							(* predefine rear side *)
							MachineCtrl.ProcessTemp.ActualJobData.SpecialTooth.VarioTooth.Distances.RearPos[0,0]	:=	1;
							MachineCtrl.ProcessTemp.ActualJobData.SpecialTooth.VarioTooth.Distances.RearPos[0,1]	:=	2;
							MachineCtrl.ProcessTemp.ActualJobData.SpecialTooth.VarioTooth.Distances.RearPos[1,0]	:=	3;
							MachineCtrl.ProcessTemp.ActualJobData.SpecialTooth.VarioTooth.Distances.RearPos[1,1]	:=	4;
							MachineCtrl.ProcessTemp.ActualJobData.SpecialTooth.VarioTooth.Distances.RearPos[2,0]	:=	5;
							MachineCtrl.ProcessTemp.ActualJobData.SpecialTooth.VarioTooth.Distances.RearPos[2,1]	:=	6;
							MachineCtrl.ProcessTemp.ActualJobData.SpecialTooth.VarioTooth.Distances.RearPos[3,0]	:=	7;
							MachineCtrl.ProcessTemp.ActualJobData.SpecialTooth.VarioTooth.Distances.RearPos[3,1]	:=	8;
							MachineCtrl.ProcessTemp.ActualJobData.SpecialTooth.VarioTooth.Distances.RearPos[4,0]	:=	9;
							MachineCtrl.ProcessTemp.ActualJobData.SpecialTooth.VarioTooth.Distances.RearPos[4,1]	:=	10;
							MachineCtrl.ProcessTemp.ActualJobData.SpecialTooth.VarioTooth.Distances.RearPos[5,0]	:=	11;
							MachineCtrl.ProcessTemp.ActualJobData.SpecialTooth.VarioTooth.Distances.RearPos[5,1]	:=	0;

							IF	( VarioCtrEnd < 5 )
								THEN
									MachineCtrl.ProcessTemp.ActualJobData.SpecialTooth.VarioTooth.Distances.RearPos[VarioCtrEnd,1]	:=	0;
							END_IF;

							FOR 	VarioCtr := 0 TO VarioCtrEnd
									DO
										VarioCtrFront1	:=	MachineCtrl.ProcessTemp.ActualJobData.SpecialTooth.VarioTooth.Distances.FrontPos[VarioCtr,0];
										VarioCtrFront2	:=	MachineCtrl.ProcessTemp.ActualJobData.SpecialTooth.VarioTooth.Distances.FrontPos[VarioCtr,1];
										VarioCtrRear1	:=	MachineCtrl.ProcessTemp.ActualJobData.SpecialTooth.VarioTooth.Distances.RearPos[VarioCtr,0];
										VarioCtrRear2	:=	MachineCtrl.ProcessTemp.ActualJobData.SpecialTooth.VarioTooth.Distances.RearPos[VarioCtr,1];

										MachineCtrl.ProcessTemp.ActualJobData.SpecialTooth.VarioTooth.Distances.Front[VarioCtr]	:=
																															VarioToothPitch[VarioCtrFront1] +
																															VarioToothPitch[VarioCtrFront2];

										MachineCtrl.ProcessTemp.ActualJobData.SpecialTooth.VarioTooth.Distances.Rear[VarioCtr]	:=
																															VarioToothPitch[VarioCtrRear1] +
																															VarioToothPitch[VarioCtrRear2];
							END_FOR;
						END_IF;
				END_IF;

				(*Transition*)
				IF	StepAction AND
					( RTrigNextStep.Q OR
					ContinousMode )
					THEN
						StepNew			:= 	1295;
						NextStepPulse	:=	FALSE;

						(* zero is the first element *)
						VarioCtr			:=	-1;
				END_IF;

	(*----------------------------------------------Calc Velocity For Automatic Process--------------------------------------------------*)

	1295:		(* action:   *)
					IF	StepActionImPulse
						THEN
							(* calc sawblade circumference *)
								SBCircumference				:=	ActualSawBlade.Diameter*PI;
								(* max feedrate chip breaker  *)
								ChipBreakerAutoXAxisMaxVelo	:=	45.0;
							(* calc velo x-axis degree/s *)
								ChipBreakerAutoVeloTemp		:=	( 360.0 * ChipBreakerAutoXAxisMaxVelo ) / SBCircumference;
								ChipBreakerXAxisVelo			:=	ChipBreakerAutoVeloTemp	;
					END_IF;

					(*Transition*)
					IF	StepAction  AND
						(NOT StepActionImPulse)
						THEN
							StepNew		:=	1297;	(*Switch On Cooling *)
					END_IF;
	(*--------------------------------------------------------Switch On Cooling ---------------------------------------------------------------*)
	1297:			(*Action*)
					IF	StepActionImPulse
						THEN
							MachineCtrl.Peripheral.ChipBreaker.Auto.Cooling.CmdOn	:=	TRUE;
							MachineCtrl.Peripheral.ChipBreaker.Auto.Cooling.CmdOff	:=	FALSE;
					END_IF;
					(*Transition*)
					IF	StepAction AND
						(NOT StepActionImPulse) AND
						MachineCtrl.State.ChipBreaker.Auto.Cooling.IsActive AND
						(NOT MachineCtrl.Peripheral.ChipBreaker.Auto.Cooling.CmdOn )
						THEN
							StepNew		:=	1300;	(*Start Process*)
					END_IF;


	(*--------------------------------------------------------------------Z-Axis Upfeed-------------------------------------------------------------*)
	1300:			(*Action*)
					IF	StepActionImPulse
						THEN
							MachineCtrl.Peripheral.ChipBreaker.Auto.DustFan.CmdOn			:=	TRUE;
							PauseAvailable												:=	TRUE;
							(*Is Demo Mode Active?*)
						(*	IF	UI.MachineSpecification.Base.DemoMode
								THEN
									ZAxisUpfeedMM	:=	-  ZAxisUpfeedMM - 1;
							END_IF;	*)
						(* set axis state for check *)
							AxisState													:=	STATE_WAIT_NEWOPERATION;
						(*	ZAxisUpfeedMM												:=	ActualJob.Infeed.TotalInfeed; *)
							ZAxisUpfeedPosition											:=	ZAxisStartPosition - (2* ZAxisUpfeedMM) ;
							ActualInfeed													:=	ActualRevolutions * MachineCtrl.ProcessTemp.ActualJobData.Job.Infeed.PartialInfeed;

							IF	( ActualJob.FeedRate.Override <= 0 )
								THEN
									ActualJob.FeedRate.Override	:=	1;
							END_IF;

							AxisCtrl[AxisNo.ZAxis].Command.OperationMode.CmdMoveAbsolut	:=	TRUE;
							AxisCtrl[AxisNo.ZAxis].Command.NominalValue.PositionMoveAbsolut	:=	ZAxisStartPosition - ZAxisUpfeedMM - 0.7;			(*= ZAxisUpfeedPosition*)
							AxisCtrl[AxisNo.ZAxis].Command.NominalValue.VeloMoveAbsolut	:=	ActualJob.FeedRate.Nominal *
																							ActualJob.FeedRate.Override;					(* velocity downfeed y-axis *)
							AxisCtrl[AxisNo.ZAxis].Command.ExternalControl.override			:=	100;
					END_IF;

					(* transition:  *)
					IF	StepAction AND
						(NOT StepActionImPulse) AND
						(* status y-axis *)
							Axis[AxisNo.ZAxis].Status.StandStill AND
							Axis[AxisNo.ZAxis].Status.InTargetPosition AND
							( AxisCtrl[AxisNo.ZAxis].feedback.state.ActualFbState = AxisState )
						THEN
							 StepNew			:= 	1305; 								(* Z-Axis Moves Down   *)
					END_IF;

	(*---------------------------------------------------------Wait For User Interaction--------------------------------------------------------------*)
		1305:		IF	StepActionImpulse
						THEN
							NextStepPulse	:=	TRUE;
					END_IF;
	
					IF	StepAction AND
						( RTrigNextStep.Q OR
						ContinousMode )
						THEN
							StepNew			:= 	1310;
							NextStepPulse	:=	FALSE;
					END_IF;

	(*--------------------------------------------------------------- Z-Axis Moves Down ---------------------------------------------------------------- *)
	1310:			(*Action*)
					IF	StepActionImPulse
						THEN
							AxisCtrl[AxisNo.ZAxis].Command.OperationMode.CmdMoveAbsolut		:=	TRUE;
							AxisCtrl[AxisNo.ZAxis].Command.NominalValue.PositionMoveAbsolut		:= 	ZAxisStartPosition ;
							AxisCtrl[AxisNo.ZAxis].Command.NominalValue.VeloMoveAbsolut		:=	3.5;
					END_IF;

					(* transition:  *)

					IF	StepAction AND
						(NOT StepActionImPulse) AND
						(* Complete movement *)
						(NOT AxisCtrl[AxisNo.ZAxis].Command.OperationMode.CmdMoveAbsolut)
						THEN
							IF	ChipBreakerfr				(*ChipBreaekerIsInFrontPosition*)
								THEN
									NominalTeeth	:=	MachineCtrl.ProcessTemp.ActualOrderStackBuffer.ActualOrder.SawBlade.NumberOfTeeth / 2;
									ActualRevolutions	:=	0;

								ELSIF	 ChipBreakerRe	(*ChipBreaekerIsInRearPosition*)
									THEN
											NominalTeeth	:=	MachineCtrl.ProcessTemp.ActualOrderStackBuffer.ActualOrder.SawBlade.NumberOfTeeth;

											ActualRevolutions	:=	1;
								END_IF;

							ActualTeeth		:=	ActualTeeth + 1;

							IF	( ActualTeeth >= NominalTeeth )
								THEN
										StepNew				:= 	10000;			(*Finish The Process*)
									ELSE
										StepNew				:= 	1350;	(*Actual Teeth <> Nominal Teeth*)
							END_IF;
								ActualInfeed			:=	ActualRevolutions * MachineCtrl.ProcessTemp.ActualJobData.Job.Infeed.PartialInfeed;
								PartialInfeed			:=	MachineCtrl.ProcessTemp.ActualJobData.Job.Infeed.PartialInfeed;
					END_IF;

	(* ---------------------------------------------------------- move x-axis ccw 2 teeth --------------------------------------------------------- *)
	1350:			(* action: *)
					IF	StepActionImPulse
						THEN
							AxisCtrl[AxisNo.XAxis].Command.OperationMode.CmdMoveAbsolut		:=	TRUE;

							IF	MachineCtrl.ProcessTemp.ActualJobData.SpecialTooth.VarioTooth.IsActive
								THEN
									VarioCtr	:=	VarioCtr + 1;

									IF	ChipBreakerRe	(*Input Variable To set The Side *)
										THEN
											AxisCtrl[AxisNo.XAxis].Command.NominalValue.PositionMoveAbsolut			:= 	Axis[AxisNo.XAxis].NcToPlc.ActPos +
																													MachineCtrl.ProcessTemp.ActualJobData.SpecialTooth.VarioTooth.Distances.Rear[VarioCtr];

										ELSIF	ChipBreakerFr
											THEN
												AxisCtrl[AxisNo.XAxis].Command.NominalValue.PositionMoveAbsolut		:= 	Axis[AxisNo.XAxis].NcToPlc.ActPos +
																													MachineCtrl.ProcessTemp.ActualJobData.SpecialTooth.VarioTooth.Distances.Front[VarioCtr];
									END_IF;

									IF	VarioCtr = VarioCtrEnd
										THEN
											VarioCtr	:=	-1;
									END_IF;

								ELSE
								(*Varion Is Inactive*)
								IF	MachineCtrl.ProcessTemp.ActualJobData.SpecialTooth.TKCompensationActive
									THEN
										IF	NoOfActTeethCompensation <> 1
											THEN
											XAxisNextPosition	:=		 Axis[AxisNo.XAxis].NcToPlc.ActPos
															         + ( 2*DegPerTeeth -
																 AxisPhasingCAM.CbaTeethDiff[NoOfActTeethCompensation] -
																 AxisPhasingCAM.CbaTeethDiff[NoOfActTeethCompensation -1] );
											ELSE
											XAxisNextPosition	:=		 Axis[AxisNo.XAxis].NcToPlc.ActPos
															         + ( 2*DegPerTeeth -
																 AxisPhasingCAM.CbaTeethDiff[1] -
																 AxisPhasingCAM.CbaTeethDiff[UI.Order.SawBlade.NumberOfTeeth] );
										END_IF;

										AxisCtrl[AxisNo.XAxis].Command.NominalValue.PositionMoveAbsolut		:= 	XAxisNextPosition;
									ELSE
										AxisCtrl[AxisNo.XAxis].Command.NominalValue.PositionMoveAbsolut		:= 	Axis[AxisNo.XAxis].NcToPlc.ActPos + ( 2 *	DegPerTeeth );
								END_IF;
							END_IF;

							AxisCtrl[AxisNo.XAxis].Command.NominalValue.VeloMoveAbsolut					:=	ChipBreakerXAxisVelo;
							AxisCtrl[AxisNo.XAxis].Command.ExternalControl.override							:=	100;
					END_IF;

					(* transition:  *)

					IF	StepAction AND
						(NOT StepActionImPulse) AND
						(* Complete movement *)
						NOT AxisCtrl[AxisNo.XAxis].Command.OperationMode.CmdMoveAbsolut
						THEN

						IF	ActualTeeth < NominalTeeth
							THEN
								NoOfActTeethCompensation		:=		NoOfActTeethCompensation   -   2 ;
								ELSIF
									(ActualTeeth = NominalTeeth)
								THEN
								;
						END_IF;

						IF	NoOfActTeethCompensation <0
							THEN
								NoOfActTeethCompensation	:=	TO_INT(UI.Order.SawBlade.NumberOfTeeth) + NoOfActTeethCompensation ;
						END_IF;

						IF	NoOfActTeethCompensation =0
							THEN
								NoOfActTeethCompensation	:=	TO_INT(UI.Order.SawBlade.NumberOfTeeth)  ;
						END_IF;

							IF 	(XAxisEndPos =AxisCtrl[AxisNo.XAxis].Command.NominalValue.PositionMoveAbsolut)		(*Check If X Reached The End Position*)
								THEN
									ContinousMode	:=	FALSE;
									StepNew		:= 	9000;														(*Check  side  finished*)
									ELSE
										IF	PauseRequested
											THEN
												ContinousMode	:=	FALSE;
												PauseAvailable	:=	FALSE;
												StepNew			:= 	30050;										(* -> pause Routine *)
											ELSE
												StepNew			:=	1300;										(*Z-Axis Upfeed*)
										END_IF;
							END_IF;
					END_IF;

	(*---------------------------------------------------------Wait For User Interaction----------------------------------------------------------*)
	9000:		IF	StepActionImpulse
					THEN
						NextStepPulse	:=	TRUE;
				END_IF;

				IF	StepAction AND
					( RTrigNextStep.Q OR
					ContinousMode )
					THEN
						StepNew			:= 	10000;
						NextStepPulse	:=	FALSE;
				END_IF;
	(*---------------------------------------------------------------End Front Side -----------------------------------------------------------------*)
	10000:		(*Transition*)
				IF	ChipBreakerFr AND
					(NOT ChipBreakerRe)
					THEN
					StepNew		:=	15000;				(*END_Front Side  *)
					XaxisEndPOsFront	:=	Axis[AxisNo.XAxis].NcToPlc.ActPos;
						ELSIF	ChipBreakerRe
					THEN
						StepNew		:=	10050;	(*Proceed to the End of Process*)
						MachineCtrl.Peripheral.ChipBreaker.Auto.DustFan.CmdOn	:=	FALSE;
				END_IF;
	(*-------------------------------------------------------Wait For User Interaction----------------------------------------------------------*)
	10050:
				IF	StepActionImpulse
					THEN
						NextStepPulse	:=	TRUE;
				END_IF;

				IF	StepAction AND
					( RTrigNextStep.Q OR
					ContinousMode )
					THEN
						StepNew			:= 	10100;
						NextStepPulse	:=	FALSE;
				END_IF;

	(* ----------------------------------------------------------- disable  Turbine  -------------------------------------------------------------- *)
	10100:		(* action *)
					IF	StepActionImPulse
						THEN
							MachineCtrl.Peripheral.ChipBreaker.Auto.Turbine.CmdOn	:=	FALSE;
							MachineCtrl.Peripheral.ChipBreaker.Auto.Turbine.CmdOff	:=	TRUE;
					END_IF;

					(* transition *)
					IF	StepAction AND
						( NOT StepActionImPulse ) AND
						( NOT MachineCtrl.Peripheral.ChipBreaker.Auto.Turbine.CmdOn )
						THEN
							StepNew		:=	10120;		(*Switch Off Fan*)
					END_IF;
	(*----------------------------------------------------------Switch Off Cooling -------------------------------------------------------*)
	10120:
					(*Action*)
					IF	StepActionImPulse
						THEN
							MachineCtrl.Peripheral.ChipBreaker.Auto.Cooling.CmdOn	:=	FALSE;
							MachineCtrl.Peripheral.ChipBreaker.Auto.Cooling.CmdOff	:=	TRUE;
					END_IF;
					(*Transition*)
					IF	StepAction AND
						(NOT StepActionImPulse) AND
						MachineCtrl.State.ChipBreaker.Auto.Cooling.IsInactive  AND
						(NOT MachineCtrl.Peripheral.ChipBreaker.Auto.Cooling.CmdOff )
						THEN
							StepNew		:=	10150;	(* ->Release Clamping *)
					END_IF;
	(*--------------------------------------------------Wait For User Interaction------------------------------------------------------------*)
	10150:		IF	StepActionImpulse
					THEN
						NextStepPulse	:=	TRUE;
				END_IF;

				IF	StepAction AND
					( RTrigNextStep.Q OR
					ContinousMode )
					THEN
						StepNew			:= 	10200;			(*Release Clamping*)
						NextStepPulse	:=	FALSE;
				END_IF;

	(*--------------------------------------------------------- Release clamping ------------------------------------------------------------- *)
	10200:		(* action *)
					IF	StepActionImPulse
						THEN
							MachineCtrl.Peripheral.ChipBreaker.Auto.Clamping.CmdClose	:=	FALSE;
							MachineCtrl.Peripheral.ChipBreaker.Auto.Clamping.CmdOpen	:=	TRUE;
					END_IF;

					(* transition:  *)
					IF	StepAction AND
						(NOT StepActionImPulse) AND
						(* clamping is opene *)
						MachineCtrl.State.ChipBreaker.Auto.Clamping.IsReleased
						THEN
							StepNew	:= 	10450;										(*Z-Axis-->Ref Pos & Saw Blade Bracket To Home Pos*)
					END_IF;
	(*--------------------------------------------Wait For User Interaction-------------------------------------------------------*)
	10450:		IF	StepActionImpulse
					THEN
						NextStepPulse	:=	TRUE;
				END_IF;

				IF	StepAction AND
					( RTrigNextStep.Q OR
					ContinousMode )
					THEN
						StepNew			:= 	10500;
						NextStepPulse	:=	FALSE;
				END_IF;
	(* ------------------------------------------------------------ sfc finished ---------------------------------------------------------- *)
	10500:		(*Action*)
					IF	 StepActionImPulse AND
						(NOT  AxisCtrl[AxisNo.ZAxis].feedback.state.DriveManagment.InHandoverPositionWindow)
						THEN
							(* Z-axis - move absolute *)
							AxisCtrl[AxisNo.ZAxis].Command.OperationMode.CmdPowerOn			:=	TRUE;
							AxisCtrl[AxisNo.ZAxis].Command.OperationMode.CmdJogHandwheel 		:=	FALSE;
							AxisCtrl[AxisNo.ZAxis].Command.OperationMode.CmdMoveAbsolut		:=	TRUE;
							AxisCtrl[AxisNo.ZAxis].Command.OperationMode.CmdCamming			:=	FALSE;
							AxisCtrl[AxisNo.ZAxis].Command.NominalValue.VeloMoveAbsolut		:=	100;
							AxisCtrl[AxisNo.ZAxis].Command.NominalValue.PositionMoveAbsolut		:=	UI.MachineSpecification.PeripheralBasic.Axis.Positions.HandOver;
							MachineCtrl.Peripheral.ChipBreaker.Auto.DustFan.CmdOn				:=	FALSE;
					END_IF;

					(*Transition : Is Z- Axis In Handover Pos?*)

					IF     	StepAction AND
					   	 (NOT StepActionImPulse) AND
						 AxisCtrl[AxisNo.ZAxis].feedback.state.DriveManagment.InHandoverPositionWindow
						THEN
							StepNew			:=	10700;							(*SB Support Bracket To Home Pos*)
							ContinousMode	:=	FALSE;
					END_IF;
	(*----------------------------------------------Wait For User Interaction------------------------------------------------*)
	10700:
					IF	StepAction AND
						NOT StepActionImPulse
						THEN
							IF	Stepper  AND
								(NOT CbaPneumatic)
								THEN
									IF	(NOT UI.MachineSpecification.Base.DemoMode)
										THEN
											StepNew		:=	10750;
										ELSE
											StepNew		:=	11000;
									END_IF;

								ELSIF	(NOT Stepper)  AND
										 CbaPneumatic
								THEN
									IF	(NOT UI.MachineSpecification.Base.DemoMode)
										THEN
											StepNew		:=	10800;
										ELSE
											StepNew		:=	11000;
									END_IF;
							END_IF;
					END_IF;

	(*----------------------------------------------------Move A-Stepper To Ref position------------------------------- *)
	10750:
				IF 	StepActionImpulse
					THEN
						AxisCtrl[AxisNo.AAxis].Command.OperationMode.CmdJog				:=	TRUE;
						AxisCtrl[AxisNo.AAxis].Command.ExternalControl.Override				:=	100;
						AxisCtrl[AxisNo.AAxis].Command.NominalValue.VeloJog				:=	0.5;
						IF	(MachineCtrl.State.ChipBreaker.Auto.AaxisActualPos <=   UI.MachineSpecification.PeripheralOptional.ChipBreaker.Notch.SBEdgeOffset)
							THEN
								AxisCtrl[AxisNo.AAxis].Command.ExternalControl.StartMinus				:=	TRUE;
								AxisCtrl[AxisNo.AAxis].Command.ExternalControl.StartPlus				:=	FALSE;;
							ELSE
								AxisCtrl[AxisNo.AAxis].Command.ExternalControl.StartMinus				:=	FALSE;
								AxisCtrl[AxisNo.AAxis].Command.ExternalControl.StartPlus				:=	TRUE;;
						END_IF;
						StartMonitoringAaxis												:=	TRUE;
				END_IF;
				(*Transition*)
				IF 	StepAction AND
					(NOT  StepActionImpulse) AND
					(MachineCtrl.State.ChipBreaker.Auto.AaxisActualPos >=  ( UI.MachineSpecification.PeripheralOptional.ChipBreaker.Notch.SBEdgeOffset  - AaxisTolerenceSlow)) AND
					(MachineCtrl.State.ChipBreaker.Auto.AaxisActualPos <=  (  UI.MachineSpecification.PeripheralOptional.ChipBreaker.Notch.SBEdgeOffset + AaxisTolerenceSlow))
					THEN
						AxisCtrl[AxisNo.AAxis].Command.ExternalControl.StartMinus				:=	FALSE;
						AxisCtrl[AxisNo.AAxis].Command.ExternalControl.StartPlus				:=	FALSE;;
						StepNew			:=	11000;
				END_IF;

	(*----------------------------------------------------Move  Cylindre To Front Position------------------------------- *)

	10800:		(*Action*)
				IF 	StepActionImpulse AND
					(NOT MachineCtrl.State.ChipBreaker.Auto.TurbinePosition.InFrontPosition)
					THEN
						MachineCtrl.Peripheral.ChipBreaker.Auto.TurbinePosition.CmdBackward	:=	FALSE;
						MachineCtrl.Peripheral.ChipBreaker.Auto.TurbinePosition.CmdForward	:=	TRUE;
				END_IF;
				(*Transition*)
				IF 	StepAction AND
					(NOT StepActionImpulse) AND
					(NOT MachineCtrl.Peripheral.ChipBreaker.Auto.TurbinePosition.CmdForward) AND
					 MachineCtrl.State.ChipBreaker.Auto.TurbinePosition.InFrontPosition
					THEN
							StepNew		:=	11000;
				END_IF;
	(*--------------------------------------CBA Swivel UnitTo Home Position----------------------------------------*)
	11000:		(*Action*)
					IF	StepActionImPulse
						THEN
							MachineCtrl.Peripheral.ChipBreaker.Auto.SwivelUnit.CmdHomePos	:=	TRUE;
							MachineCtrl.Peripheral.ChipBreaker.Auto.SwivelUnit.CmdWorkPos	:=	FALSE;
							StartMonitoringAaxis											:=	FALSE;
					END_IF;
					(*Transition*)
					IF 	StepAction AND
						(NOT StepActionImPulse) AND
						MachineCtrl.State.ChipBreaker.Auto.SwivelUnit.InHomePosition
						THEN
							StepNew		:=	11010;	(*Wait for New Operation*)
					END_IF;

	(*----------------------------------------------------Wait For User Interaction-----------------------------------------------*)
	11010:
					IF	StepActionImpulse
						THEN
							NextStepPulse	:=	TRUE;
					END_IF;
	
					IF	StepAction AND
						( RTrigNextStep.Q OR
						ContinousMode )
						THEN
							StepNew			:= 	15000;
							NextStepPulse	:=	FALSE;
					END_IF;
	(*---------------------------------------Step 10 : Wait for New Operation-------------------------------------------*)

	15000:		(* transition *)
					IF	StepAction AND
						(NOT StepActionImPulse)
							THEN
								IF 	ChipBreakerRe
									THEN
										StepNew				:= 	16000;			(*Wait For New Operation*)
										MachineCtrl.Peripheral.ChipBreaker.Auto.LowSpeedMonitoring.IsDeactivated	:=	FALSE;
										Done				:=	TRUE;
										Start					:=	FALSE;
										ChipBreakerFr		:=	TRUE;
										ChipBreakerRe		:=	FALSE;
									ELSIF 	ChipBreakerFr
										THEN
										ChipBreakerFr	:=	FALSE;
										ChipBreakerRe	:=	TRUE;
										IF	Stepper AND
											(NOT CbaPneumatic)
											THEN
												StepNew			:= 	950;		(*Start With The Rear Side*)
											ELSIF	CbaPneumatic AND
													(NOT Stepper)
											THEN
												StepNew			:= 	990;
										END_IF;
										Done	:=	FALSE;
								END_IF;
					END_IF;

	(*---------------------------------------Wait For User Interaction---------------------------------------------------------*)
	16000:		IF	StepActionImpulse
					THEN
						NextStepPulse	:=	TRUE;
				END_IF;

				IF	StepAction AND
					( RTrigNextStep.Q OR
					ContinousMode )
					THEN
						StepNew			:= 	10;
						NextStepPulse	:=	FALSE;
				END_IF;

	(*--##################################---ERROR-###################################- *)

	25000:		(*Action*)
				IF	 StepActionImPulse
					THEN
						MachineCtrl.Peripheral.ChipBreaker.Auto.DustFan.CmdOn			:=	FALSE;
						AxisCtrl[AxisNo.AAxis].Command.ExternalControl.StartPlus			:=	FALSE;
						AxisCtrl[AxisNo.AAxis].Command.ExternalControl.StartMinus			:=	FALSE;		(*Stop Moving   A-Axis*)
						ErrorOut			:=	TRUE;
				END_IF;
				(*Transition*)

				IF 	StepAction AND
					(NOT StepActionImPulse)
					THEN
						StepNew		:=	0;
						ErrorOut		:=	FALSE;
				END_IF;
	(* ####################################### pause sfc ################################ *)

	(*-----------------------------------------------------------Wait For User Interaction------------------------------------------------*)
	30050:
				 IF	StepActionImpulse
					THEN
						NextStepPulse	:=	TRUE;
				END_IF;

				IF	StepAction AND
					( RTrigNextStep.Q OR
					ContinousMode )
					THEN
						StepNew			:= 	30100;		(*Release Clamping*)
						NextStepPulse	:=	FALSE;
				END_IF;

	(*--------------------------------------------------------------Release Clamping-----------------------------------------------------*)
	30100:
					(*Action*)
				IF	StepActionImPulse
					THEN
						MachineCtrl.Peripheral.ChipBreaker.Auto.Clamping.CmdClose	:=	FALSE;
						MachineCtrl.Peripheral.ChipBreaker.Auto.Clamping.CmdOpen	:=	TRUE;
				END_IF;

				(* transition:  *)

				IF	StepAction AND
					(NOT StepActionImPulse) AND
					MachineCtrl.State.ChipBreaker.Auto.Clamping.IsReleased
					THEN
						StepNew	:= 	30200;					(*Z Axis Move   down 100 MM*)
				END_IF;
	(* ----------------------------------------------------- wait for user interaction  ---------------------------------------------------- *)
	30200:
				IF	StepActionImpulse
					THEN
						NextStepPulse	:=	TRUE;
				END_IF;

				IF	StepAction AND
					( RTrigNextStep.Q OR
					ContinousMode )
					THEN
						StepNew			:= 	30250;
						NextStepPulse	:=	FALSE;
				END_IF;
	(* ------------------------------------------------- sfc Paused: move Z-axisDown ------------------------------------------------- *)

	30250	:	(* action: move z-axis down  *)
				IF	StepActionImPulse
					THEN
					(* set axis state for check *)
						AxisState	:=	STATE_WAIT_NEWOPERATION;
					(* move y-axis to reference point *)
						AxisCtrl[AxisNo.ZAxis].Command.OperationMode.CmdPowerOn					:=	TRUE;
						AxisCtrl[AxisNo.ZAxis].Command.OperationMode.CmdMoveAbsolut				:=	TRUE;
						AxisCtrl[AxisNo.ZAxis].Command.NominalValue.PositionMoveAbsolut				:=	Axis[AxisNo.ZAxis].NcToPlc.ActPos	+100;
						AxisCtrl[AxisNo.ZAxis].Command.NominalValue.VeloMoveAbsolut				:=	30;
						MachineCtrl.Peripheral.ChipBreaker.Auto.DustFan.CmdOn						:=	FALSE;
				END_IF;

				(* transition *)
				IF	StepAction AND
					(NOT StepActionImPulse) AND
					(* status Z-axis *)
					Axis[AxisNo.ZAxis].Status.StandStill AND
					Axis[AxisNo.ZAxis].Status.InTargetPosition AND
					( NOT AxisCtrl[AxisNo.ZAxis].Command.OperationMode.CmdMoveAbsolut ) AND
					( AxisCtrl[AxisNo.ZAxis].feedback.state.ActualFbState = AxisState )
					THEN
						StepNew		:= 30300;															(*Turbine Off*)
				END_IF;

	(* ---------------------------------------------------- wait for user interaction  ------------------------------------------------------------ *)
	30300:		IF	StepActionImpulse
					THEN
						NextStepPulse	:=	TRUE;
				END_IF;

				IF	StepAction AND
					( RTrigNextStep.Q OR
					ContinousMode )
					THEN
						StepNew			:= 	30350;	(*Turbine Off*)
						NextStepPulse	:=	FALSE;
				END_IF;

	(* --------------------------------------------------------------- Turbine Off --------------------------------------------------------------------- *)
	30350	:	(* action:   *)
				IF	StepActionImPulse
					THEN
						MachineCtrl.Peripheral.ChipBreaker.Auto.Turbine.CmdOn	:=	FALSE;
						MachineCtrl.Peripheral.ChipBreaker.Auto.Turbine.CmdOff	:=	TRUE;
				END_IF;
				(* transition: *)
				IF	StepAction AND
					( NOT StepActionImPulse ) AND
					( NOT MachineCtrl.Peripheral.ChipBreaker.Auto.Turbine.CmdOn )AND
					(NOT MachineCtrl.State.ChipBreaker.Auto.Turbine.IsActive)			(*Turbine Is Inactive*)
					THEN
							StepNew		:=	30370	;
				END_IF;

	(*-------------------------------------------------------Switch Off Cooling --------------------------------------------------------------------*)
	30370:
				(*Action*)
				IF	StepActionImPulse
					THEN
						MachineCtrl.Peripheral.ChipBreaker.Auto.Cooling.CmdOn	:=	FALSE;
						MachineCtrl.Peripheral.ChipBreaker.Auto.Cooling.CmdOff	:=	TRUE;
				END_IF;
				(*Transition*)
				IF	StepAction AND
					(NOT StepActionImPulse) AND
					MachineCtrl.State.ChipBreaker.Auto.Cooling.IsInactive  AND
					(NOT MachineCtrl.Peripheral.ChipBreaker.Auto.Cooling.CmdOff )
					THEN
						StepNew		:=	30400;	(* ->deactivate axis x/z *)
				END_IF;
	(* ------------------------------------------------------ wait for user interaction  -------------------------------------------------------------- *)
	30400:
				IF	StepActionImpulse
					THEN
						NextStepPulse	:=	TRUE;
				END_IF;

				IF	StepAction AND
					( RTrigNextStep.Q OR
					ContinousMode )
					THEN
						StepNew			:= 	30450;
						NextStepPulse	:=	FALSE;
				END_IF;
	(*---------------------------------------------------------------Desable X/Z Axis-----------------------------------------------------------------*)
	30450:
				(* action:   *)
				IF	StepActionImPulse
					THEN
						(* set axis state for check *)
							AxisState	:=	STATE_INIT;
						(* x-axis - disable *)
							AxisCtrl[AxisNo.XAxis].Command.OperationMode.CmdPowerOn			:=	FALSE;
							AxisCtrl[AxisNo.XAxis].Command.OperationMode.CmdMoveAbsolut		:=	FALSE;
							AxisCtrl[AxisNo.XAxis].Command.OperationMode.CmdCamming			:=	FALSE;
						(* z-axis - disable *)
							AxisCtrl[AxisNo.ZAxis].Command.OperationMode.CmdPowerOn			:=	FALSE;
							AxisCtrl[AxisNo.ZAxis].Command.OperationMode.CmdMoveAbsolut		:=	FALSE;
							AxisCtrl[AxisNo.ZAxis].Command.OperationMode.CmdCamming			:=	FALSE;
				END_IF;
				(* transition:  *)
				IF	StepAction AND
					(NOT StepActionImPulse) AND
					(* status x-axis *)
						Axis[AxisNo.XAxis].Status.Disabled AND
						( AxisCtrl[AxisNo.XAxis].feedback.state.ActualFbState = AxisState ) AND
					(* status z-axis *)
						Axis[AxisNo.ZAxis].Status.Disabled AND
						( AxisCtrl[AxisNo.ZAxis].feedback.state.ActualFbState = AxisState )
						THEN
							StepNew		:= 	30460;			(*User Interaction*)
				END_IF;
	(* ------------------------------------------------------------- wait for user interaction  -------------------------------------------------------- *)
	30460:
				IF	StepActionImpulse
					THEN
						NextStepPulse	:=	TRUE;
				END_IF;

				IF	StepAction AND
					( RTrigNextStep.Q OR
					ContinousMode )
					THEN
						StepNew			:= 	30470;		(* -> Activate Safety State*)
						NextStepPulse	:=	FALSE;
				END_IF;
	(* -------------------------------------------------------- Activate Safety State -------------------------------------------------------------- *)
	30470:				(*Action*)
				IF	StepActionImPulse
					THEN
					(* Enable safe state  *)
						MachineCtrl.Peripheral.SafetyState.CmdActivate	:=	TRUE;
						MachineCtrl.State.GrindingWheel.PauseIsActive	:=	TRUE;
				END_IF;
				(* transition:  *)
				IF	StepAction AND
					(NOT StepActionImPulse) AND
					(* state safety state *)
					( NOT MachineCtrl.Peripheral.SafetyState.CmdActivate ) AND
					MachineCtrl.state.SafetyState.unit.IsActive
					THEN
						StepNew		:=	30500;
				END_IF;

	(*--------------------------------------------------------------------Set Event----------------------------------------------------------------------*)
				(*Action*)
	30500:
				IF	StepActionImPulse
					THEN
				(* set Event *)
						MachineCtrl.ProcessControl.Event.No		:=	EvNoStartStop;
						MachineCtrl.ProcessControl.Event.En		:=	TRUE;
						MachineCtrl.ProcessControl.Event.SId	:=	EvEventSourceId;
						MachineCtrl.ProcessControl.Event.Class	:=	TcEventClassMessage;
						MachineCtrl.Peripheral.Buzzer.Unit.CmdOn:=	TRUE;
				END_IF;
				(*Transition*)
				IF	StepAction AND
					(NOT StepActionImPulse)
					THEN
						StepNew		:=	30520;
				END_IF;

	(* --------------------------------------------------------- wait for user interaction  ---------------------------------------------------------- *)
	30520:		IF	StepActionImpulse
					THEN
						NextStepPulse	:=	TRUE;
				END_IF;

				IF	StepAction AND
					( RTrigNextStep.Q OR
					ContinousMode )
					THEN
						MachineCtrl.Peripheral.ChipBreaker.Auto.DustFan.CmdOn					:=	FALSE;
						MachineCtrl.Peripheral.ChipBreaker.Auto.LowSpeedMonitoring.IsDeactivated	:=	FALSE;
						StepNew			:= 	30550;	(*Deactivate Safety  State *)
						NextStepPulse	:=	FALSE;
						Paused			:=	TRUE;
				END_IF;
	(* -----------------------------------------------------Deactivate Safety State---------------------------------------------------------- *)
	30550:			(* action:   *)
				IF	MachineCtrl.state.SafetyState.unit.IsActive
					THEN
						MachineCtrl.Peripheral.ChipBreaker.Auto.LowSpeedMonitoring.IsDeactivated	:=	FALSE;
						IF	MachineStateSharpenerDoorIsClosed AND
							AutomaticMode
							THEN
								(* Disable safe state  *)
								MachineCtrl.Peripheral.SafetyState.CmdDeactivate	:=	TRUE;
								MachineCtrl.State.GrindingWheel.PauseIsActive	:=	FALSE;
							ELSE
								(* Disable safe state  *)
								MachineCtrl.Peripheral.SafetyState.CmdDeactivate	:=	FALSE;
								MachineCtrl.Peripheral.SafetyState.CmdActivate	:=	TRUE;
								MachineCtrl.State.GrindingWheel.PauseIsActive	:=	TRUE;
						END_IF;
				END_IF;

				TONWaitSafetyStatePause( IN  	:=  	StepAction AND
												( NOT MachineCtrl.Peripheral.SafetyState.CmdDeactivate ) AND
												( NOT MachineCtrl.state.SafetyState.unit.IsActive ),
										 PT 	:= 	TIME#50ms);

				(* transition:  *)
				IF	StepAction AND
					(NOT StepActionImPulse) AND
					(* state safety state *)
						( NOT MachineCtrl.Peripheral.SafetyState.CmdDeactivate ) AND
						( NOT MachineCtrl.state.SafetyState.unit.IsActive ) AND
						TONWaitSafetyStatePause.Q (* AND
					StartSwitch *)
					THEN
						MachineCtrl.ProcessControl.Event.No		:=	0;
						MachineCtrl.ProcessControl.Event.En		:=	FALSE;
						StepNew								:= 	30600;	(*Turbine On*)
				END_IF;

	(* ----------------------------------------------------------- wait for user interaction  ------------------------------------------------ *)
	30600:		IF	StepActionImpulse
					THEN
						MachineCtrl.Peripheral.ChipBreaker.Auto.LowSpeedMonitoring.IsDeactivated	:=		TRUE;
						NextStepPulse	:=	TRUE;
				END_IF;

				IF	StepAction AND
					( RTrigNextStep.Q OR
					ContinousMode )
					THEN
						StepNew			:= 	30650;			(*Activate Turbine *)
						NextStepPulse	:=	FALSE;
				END_IF;

	(*------------------------------------------------------------------Turbine On--------------------------------------------------------------------*)
	30650:			(*Action*)
				IF	 StepActionImPulse
						THEN
							MachineCtrl.Peripheral.ChipBreaker.Auto.Turbine.CmdOn	:=	TRUE;
							MachineCtrl.Peripheral.ChipBreaker.Auto.Turbine.CmdOff	:=	FALSE;
				END_IF;
				(*Transition: Is the  Turbine On? *)
				IF	 StepAction 	AND
					 (NOT StepActionImPulse) AND
				    	  MachineCtrl.State.ChipBreaker.Auto.Turbine.IsActive
					THEN
						StepNew		:=	30660;		(*Switch On Cooling Fan*)
				END_IF;

	(*---------------------------------------------------- Switch On Cooling -------- --------------------------------------------------------------*)

	30660:
			(*Action*)
				IF	StepActionImPulse
					THEN
						MachineCtrl.Peripheral.ChipBreaker.Auto.Cooling.CmdOn	:=	TRUE;
						MachineCtrl.Peripheral.ChipBreaker.Auto.Cooling.CmdOff	:=	FALSE;
				END_IF;
				(*Transition*)
				IF	StepAction AND
					(NOT StepActionImPulse) AND
					MachineCtrl.State.ChipBreaker.Auto.Cooling.IsActive AND
					(NOT MachineCtrl.Peripheral.ChipBreaker.Auto.Cooling.CmdOn )
					THEN
						StepNew		:=	30670;	(*Start Process*)
				END_IF;

	(* ---------------------------------------------------- wait for user interaction  ------------------------------------------------------------ *)
	30670:
				IF	StepActionImpulse
					THEN
						NextStepPulse	:=	TRUE;
				END_IF;

				IF	StepAction AND
					( RTrigNextStep.Q OR
					ContinousMode )
					THEN
						StepNew			:= 	30680;			(*Open Clamping*)
						NextStepPulse	:=	FALSE;
				END_IF;
	(* ------------------------------------------------------- sfc Paused: Open Clamping ---------------------------------------------------- *)
	30680	:		(*Action*)
				IF	StepActionImPulse
					THEN
						MachineCtrl.Peripheral.ChipBreaker.Auto.Clamping.CmdClose	:=	FALSE;
						MachineCtrl.Peripheral.ChipBreaker.Auto.Clamping.CmdOpen	:=	TRUE;
				END_IF;
				(* transition:  *)
				IF	StepAction AND
					(NOT StepActionImPulse) AND
					MachineCtrl.State.ChipBreaker.Auto.Clamping.IsReleased
				THEN
						StepNew	:= 	30700;			(*Move Z To Start Pos*)
				END_IF;

	(* ----------------------------------------------------------- wait for user interaction  --------------------------------------------------------- *)
	30700:		IF	StepActionImpulse
					THEN
						NextStepPulse	:=	TRUE;
				END_IF;

				IF	StepAction AND
					( RTrigNextStep.Q OR
					ContinousMode )
					THEN
						StepNew			:= 	30710;
						NextStepPulse	:=	FALSE;
				END_IF;

	(*----------------------------------------------------------Move Z Axis To Start Pos-----------------------------------------------------------*)
	30710:
					(*Action*)
				IF	StepActionImPulse
				THEN
					AxisState	:=	STATE_WAIT_NEWOPERATION;
				(* Z-axis - move absolute *)
					AxisCtrl[AxisNo.ZAxis].Command.OperationMode.CmdPowerOn			:=	TRUE;
					AxisCtrl[AxisNo.ZAxis].Command.OperationMode.CmdJogHandwheel 		:=	FALSE;
					AxisCtrl[AxisNo.ZAxis].Command.OperationMode.CmdMoveAbsolut		:=	TRUE;
					AxisCtrl[AxisNo.ZAxis].Command.OperationMode.CmdCamming			:=	FALSE;
					AxisCtrl[AxisNo.ZAxis].Command.NominalValue.PositionMoveAbsolut		:=	ZAxisStartPosition;			(* Startposition y-axis *)
					AxisCtrl[AxisNo.ZAxis].Command.NominalValue.VeloMoveAbsolut		:=	15;						(* velocity Startpos z-axis *)
					AxisCtrl[AxisNo.ZAxis].Command.ExternalControl.override				:=	100;
				END_IF;

				(*Transition : Is /Z Axis in Start Position*)
				IF 	StepAction AND
					(NOT StepActionImPulse) AND
					(* status Z-axis *)
						Axis[AxisNo.ZAxis].Status.StandStill AND
						Axis[AxisNo.ZAxis].Status.InTargetPosition AND
						( NOT AxisCtrl[AxisNo.ZAxis].Command.OperationMode.CmdMoveAbsolut ) AND
						( AxisCtrl[AxisNo.ZAxis].feedback.state.ActualFbState = AxisState )
				THEN
					StepNew		:=	30800;		(*Clamping*)
				END_IF;

	(* ---------------------------------------------------- wait for user interaction  ------------------------------------------------------------- *)
	30800:
				IF	StepActionImpulse
					THEN
						NextStepPulse	:=	TRUE;
				END_IF;

				IF	StepAction AND
					( RTrigNextStep.Q OR
					ContinousMode )
					THEN
						StepNew			:= 	30860; (*Close Clamping*)
						NextStepPulse	:=	FALSE;
				END_IF;
	(*-----------------------------------------------------------------Close Klamping------------------------------------------------------------*)
	30860:
				(*Action*)
				IF	StepActionImPulse
					THEN
						MachineCtrl.Peripheral.ChipBreaker.Auto.Clamping.CmdClose	:=	TRUE;
						MachineCtrl.Peripheral.ChipBreaker.Auto.Clamping.CmdOpen	:=	FALSE;
				END_IF;

				WaitAfterPause(IN:=	StepAction AND
									(NOT StepActionImPulse) AND
									(* clamping is open *)
									MachineCtrl.State.ChipBreaker.Auto.Clamping.ClampingIsOn ,
									PT:=TIME#2s , Q=> , ET=> );

				(* transition:  *)
				IF	StepAction AND
					(NOT StepActionImPulse) AND
					(* clamping is open *)
					MachineCtrl.State.ChipBreaker.Auto.Clamping.ClampingIsOn AND
					WaitAfterPause.Q
					THEN
						StepNew				:=	30910 	;	(*30910/Pause Step*)
						Paused				:=	FALSE;
						PauseRequested		:=	FALSE;
				END_IF;
	(* --------------------------------------------------------- wait for user interaction  ------------------------------------------------------------ *)
	30910:
				IF	StepActionImpulse
					THEN
						NextStepPulse	:=	TRUE;
				END_IF;
	
				IF	StepAction AND
					( RTrigNextStep.Q OR
					ContinousMode )
					THEN
						StepNew			:= 	30915; 					(*Enable X/Z Axis*)
						NextStepPulse	:=	FALSE;
				END_IF;

	(*-------------------------------------------------------------------Enable Axis---------------------------------------------------------------------*)
	30915:	(*Action*)
			IF	StepActionImPulse
				THEN
				(* set axis state for check *)
					AxisState	:=	STATE_WAIT_NEWOPERATION;
				(* x-axis - Enable *)
					AxisCtrl[AxisNo.XAxis].Command.OperationMode.CmdPowerOn			:=	TRUE;
					AxisCtrl[AxisNo.XAxis].Command.OperationMode.CmdMoveAbsolut		:=	FALSE;
					AxisCtrl[AxisNo.XAxis].Command.OperationMode.CmdCamming			:=	FALSE;
					AxisCtrl[AxisNo.XAxis].Command.ExternalControl.override				:=	100;
				(* z-axis - Enable *)
					AxisCtrl[AxisNo.ZAxis].Command.OperationMode.CmdPowerOn			:=	TRUE;
					AxisCtrl[AxisNo.ZAxis].Command.OperationMode.CmdMoveAbsolut		:=	FALSE;
					AxisCtrl[AxisNo.ZAxis].Command.OperationMode.CmdCamming			:=	FALSE;
					AxisCtrl[AxisNo.ZAxis].Command.ExternalControl.override				:=	100;
			END_IF;

			(* transition: axis are Enabled? *)
			IF	StepAction AND
				(NOT StepActionImPulse) AND
				(* status x-axis *)
					(NOT Axis[AxisNo.XAxis].Status.Disabled) AND
					Axis[AxisNo.XAxis].Status.StandStill AND
					( AxisCtrl[AxisNo.XAxis].feedback.state.ActualFbState = AxisState ) AND
				(* status Z-axis *)
					(NOT Axis[AxisNo.ZAxis].Status.Disabled) AND
					Axis[AxisNo.ZAxis].Status.StandStill AND
					( AxisCtrl[AxisNo.ZAxis].feedback.state.ActualFbState = AxisState ) AND
				(* stop switch not pressed *)
					(PauseSwitchActive)
				THEN
					StepNew	:= 	30920;								(* -> User Interaction *)
			END_IF;

	(* -------------------------------------------------------------- wait for user interaction  ----------------------------------------------------- *)
	30920:
			IF	StepActionImpulse
				THEN
					NextStepPulse	:=	TRUE;
			END_IF;

			IF	StepAction AND
				( RTrigNextStep.Q OR
				ContinousMode )
				THEN
					MachineCtrl.Peripheral.ChipBreaker.Auto.DustFan.CmdOn	:=	TRUE;
					StepNew			:= 	1300; 			(*Pause-Step : X/Z Start Pos , Or 1300 : Z-Axis Upfeed*)
					NextStepPulse	:=	FALSE;
			END_IF;
	(*##########################################STOP#########################################*)

	(*-------------------------------------------------------------------Stop Z-Axis--------------------------------------------------------------------*)

	31000:	(*Action*)
			IF	 StepActionImPulse
				THEN
					(* set axis state for check *)
					AxisState	:=	STATE_WAIT_NEWOPERATION;
					(* Z-axis - move absolute Stopped *)
					AxisCtrl[AxisNo.ZAxis].Command.OperationMode.CmdPowerOn			:=	TRUE;;
					AxisCtrl[AxisNo.ZAxis].Command.OperationMode.CmdJogHandwheel 		:=	FALSE;
					AxisCtrl[AxisNo.ZAxis].Command.OperationMode.CmdMoveAbsolut		:=	FALSE;
					AxisCtrl[AxisNo.ZAxis].Command.OperationMode.CmdCamming			:=	FALSE;
					AxisCtrl[AxisNo.ZAxis].Command.NominalValue.VeloMoveAbsolut		:=	(*50;*)0;
					AxisCtrl[AxisNo.ZAxis].Command.NominalValue.PositionMoveAbsolut		:=	UI.MachineSpecification.PeripheralBasic.Axis.Positions.HandOver;
					MachineCtrl.Peripheral.ChipBreaker.Auto.DustFan.CmdOn				:=	FALSE;
					StartMonitoringAaxis												:=	FALSE;
			END_IF;
				(*Transition Z-Axis *)
				IF     	StepAction AND
				   	 (NOT StepActionImPulse) AND
					(AutomaticMode OR MachineCtrl.State.Mode.InitSetUp.IsActive  ) AND
					(* status Z-axis *)
					(NOT Axis[AxisNo.ZAxis].Status.Disabled) AND
					Axis[AxisNo.ZAxis].Status.StandStill AND
					( AxisCtrl[AxisNo.ZAxis].feedback.state.ActualFbState = AxisState )
					THEN
						StepNew		:= 31020	;		(*Stop Turbine*)
				END_IF;
	(*-------------------------------------------------------------Wait For User Interaction-----------------------------------------------------------*)
	31020:
			IF	StepActionImpulse
				THEN
					NextStepPulse	:=	TRUE;
			END_IF;

			IF	StepAction AND
				( RTrigNextStep.Q OR
				ContinousMode )
				THEN
					StepNew			:= 	31030; 				(*Stop Z-Axis*)
					NextStepPulse	:=	FALSE;
					StartWaitAaxis	:=	TRUE;
			END_IF;

	(*-----------------------------------------------------------------Turbine Off----------------------------------------------------------------------------*)
	31030:
			(* action:   *)
			IF	StepActionImPulse
				THEN
					MachineCtrl.Peripheral.ChipBreaker.Auto.Turbine.CmdOn	:=	FALSE;
					MachineCtrl.Peripheral.ChipBreaker.Auto.Turbine.CmdOff	:=	TRUE;
			END_IF;

			IF	StepAction AND
				( NOT StepActionImPulse ) AND
				( NOT MachineCtrl.Peripheral.ChipBreaker.Auto.Turbine.CmdOn )AND
				(NOT MachineCtrl.State.ChipBreaker.Auto.Turbine.IsActive)
				THEN
					StepNew		:=	31100;									(* Switch Off Cooling Fan *)
			END_IF;
	(*-----------------------------------------------------------Switch Off Cooling ----------------------------------------------------------------------*)
	31100:
			(*Action*)
			IF	StepActionImPulse
				THEN
					MachineCtrl.Peripheral.ChipBreaker.Auto.Cooling.CmdOn	:=	FALSE;
					MachineCtrl.Peripheral.ChipBreaker.Auto.Cooling.CmdOff	:=	TRUE;
					StartWaitAaxis										:=	FALSE;
			END_IF;
			(*Transition*)
			IF	StepAction AND
				(NOT StepActionImPulse) AND
				MachineCtrl.State.ChipBreaker.Auto.Cooling.IsInactive  AND
				(NOT MachineCtrl.Peripheral.ChipBreaker.Auto.Cooling.CmdOff )
				THEN
					StepNew		:=	31300;			(*Release Clamping*)
			END_IF;
	(*------------------------------------------------------------Wait For User Interaction-------------------------------------------------------------*)
	31300:
			IF	StepActionImpulse
				THEN
					NextStepPulse	:=	TRUE;
			END_IF;

			IF	StepAction AND
				( RTrigNextStep.Q OR
				ContinousMode )
				THEN
					StepNew			:= 	31320; 				(*Release Clamping*)
					NextStepPulse	:=	FALSE;
			END_IF;
	(*---------------------------------------------------------------------Move Z-Axis Dwn 5 MM-----------------------------------------------------------      *)
	31320:
			IF 	StepActionImPulse
				THEN
					AxisState																:=	STATE_WAIT_NEWOPERATION;
					AxisCtrl[AxisNo.ZAxis].Command.OperationMode.CmdPowerOn					:=	TRUE;;
					AxisCtrl[AxisNo.ZAxis].Command.OperationMode.CmdMoveAbsolut				:=	TRUE;
					AxisCtrl[AxisNo.ZAxis].Command.ExternalControl.override						:=	100;
					AxisCtrl[AxisNo.ZAxis].Command.OperationMode.CmdMoveAbsolutTouchProbe	:=	FALSE;
					AxisCtrl[AxisNo.ZAxis].Command.NominalValue.PositionMoveAbsolut				:=	Axis[AxisNo.ZAxis].NcToPlc.ActPos + 5;
					AxisCtrl[AxisNo.ZAxis].Command.NominalValue.VeloMoveAbsolut				:=	2;
			END_IF;
			(*Transition*)
			IF	StepAction AND
				NOT StepActionImPulse  AND
				(* status z-axis *)
				( NOT Axis[AxisNo.ZAxis].Status.Disabled ) AND
				Axis[AxisNo.ZAxis].Status.InTargetPosition AND
				Axis[AxisNo.ZAxis].Status.StandStill	AND
				( NOT AxisCtrl[AxisNo.ZAxis].Command.OperationMode.CmdMoveAbsolut )AND
				( AxisCtrl[AxisNo.ZAxis].feedback.state.ActualFbState = AxisState )
				THEN
					AxisCtrl[AxisNo.ZAxis].Command.OperationMode.CmdMoveAbsolut	:=	FALSE;
					StepNew		:=	31350;
			END_IF
	(*-------------------------------------------------------------------Release clamping----------------------------------------------------------------*)
	31350:
			(*Action*)
			IF	StepActionImPulse AND
				(NOT MachineCtrl.State.ChipBreaker.Auto.Clamping.IsReleased)
				THEN
					MachineCtrl.Peripheral.ChipBreaker.Auto.Clamping.CmdClose	:=	FALSE;
					MachineCtrl.Peripheral.ChipBreaker.Auto.Clamping.CmdOpen	:=	TRUE;
			END_IF;

			(* transition:  *)
			IF	StepAction AND
				(NOT StepActionImPulse) AND
				MachineCtrl.State.ChipBreaker.Auto.Clamping.IsReleased
			THEN
					StepNew	:= 	31360;					(*Z Axis  down*)
			END_IF;

	(*---------------------------------------------------------------Wait For User Interaction--------------------------------------------------------------*)
	31360:
			IF	StepActionImpulse
				THEN
					NextStepPulse	:=	TRUE;
			END_IF;

			IF	StepAction AND
				( RTrigNextStep.Q OR
				ContinousMode )
				THEN
					StepNew			:= 	31370; 				(*Move Z -axis To Handover Position*)
					NextStepPulse	:=	FALSE;
			END_IF;
	(*-----------------------------------------------------------Move Z-Axis To handover Position-----------------------------------------------------*)
	31370:
			(*Action*)
			IF	 StepActionImPulse AND
				(NOT  AxisCtrl[AxisNo.ZAxis].feedback.state.DriveManagment.InHandoverPositionWindow)
				THEN
					(* Z-axis - move absolute *)
					AxisCtrl[AxisNo.ZAxis].Command.OperationMode.CmdPowerOn			:=	TRUE;
					AxisCtrl[AxisNo.ZAxis].Command.OperationMode.CmdJogHandwheel 		:=	FALSE;
					AxisCtrl[AxisNo.ZAxis].Command.OperationMode.CmdMoveAbsolut		:=	TRUE;
					AxisCtrl[AxisNo.ZAxis].Command.OperationMode.CmdCamming			:=	FALSE;
					AxisCtrl[AxisNo.ZAxis].Command.NominalValue.VeloMoveAbsolut		:=	100;
					AxisCtrl[AxisNo.ZAxis].Command.NominalValue.PositionMoveAbsolut		:=	UI.MachineSpecification.PeripheralBasic.Axis.Positions.HandOver;
			END_IF;
				(*Transition : Is Z- Axis In Handover Pos?*)
				IF     	StepAction AND
				   	 (NOT StepActionImPulse) AND
					 AxisCtrl[AxisNo.ZAxis].feedback.state.DriveManagment.InHandoverPositionWindow
					THEN
						IF	Stepper  AND
							(NOT CbaPneumatic)
							THEN
								StepNew	:=	31375;
						ELSIF	CbaPneumatic AND
								(NOT Stepper)
							THEN
								StepNew	:=	31400;		(*CbaPneumatic To front Position*)
						END_IF;
				END_IF;

	(*----------------------------------------------------------------Move A-Stepper To Ref Position----------------------------------------------------------------------*)
	31375:
			IF 	StepAction AND
				(NOT  StepActionImpulse)
				THEN
					AxisCtrl[AxisNo.AAxis].Command.ExternalControl.StartMinus				:=	FALSE;
					AxisCtrl[AxisNo.AAxis].Command.ExternalControl.StartPlus				:=	FALSE;;
					StepNew					:=	31450;
					StartMonitoringAaxis		:=	FALSE;
			END_IF;
	(*-----------------------------------------------Cylindre To Front Position---------------------------------------------------------------------*)
	31400:
			(*Action*)
			IF 	StepActionImpulse AND
				(NOT MachineCtrl.State.ChipBreaker.Auto.TurbinePosition.InFrontPosition)
				THEN
					MachineCtrl.Peripheral.ChipBreaker.Auto.TurbinePosition.CmdBackward	:=	FALSE;
					MachineCtrl.Peripheral.ChipBreaker.Auto.TurbinePosition.CmdForward	:=	TRUE;
			END_IF;
			(*Transition*)
			IF 	StepAction AND
				(NOT StepActionImpulse) AND
				((NOT MachineCtrl.Peripheral.ChipBreaker.Auto.TurbinePosition.CmdForward) AND
				 MachineCtrl.State.ChipBreaker.Auto.TurbinePosition.InFrontPosition AND
				CbaPneumatic) OR Stepper
				THEN
					StepNew		:=	31450;						(*chipBreaker SU---> HomePos*)
			END_IF;
	(*-------------------------------------------------------Chip Breaker Swivel Unit To Home Position------------------------------------------*)
	31450:
			(*Action *)
			IF 	StepActionImpulse AND
				(NOT MachineCtrl.State.ChipBreaker.Auto.SwivelUnit.InHomePosition)
				THEN
					MachineCtrl.Peripheral.ChipBreaker.Auto.SwivelUnit.CmdHomePos	:=	TRUE;
					MachineCtrl.Peripheral.ChipBreaker.Auto.SwivelUnit.CmdWorkPos	:=	FALSE;
			END_IF;

			(*Transition : Is Chip Breaker In Work Position?*)

			IF 	StepAction AND
			   	 (NOT StepActionImPulse) AND
			     	MachineCtrl.State.ChipBreaker.Auto.SwivelUnit.InHomePosition
				THEN
					StepNew		:=	31500;					(*STOP*)
			END_IF;
	(*--------------------------------------------------------------Wait For User Interaction----------------------------------------------------------------------*)
	31500:
			IF	StepActionImpulse
				THEN
					NextStepPulse	:=	TRUE;
			END_IF;

			IF	StepAction AND
				( RTrigNextStep.Q OR
				ContinousMode )
				THEN
					StepNew			:= 	31550; 				(*Move Z -axis To Handover Position*)
					NextStepPulse	:=	FALSE;
			END_IF;
		(*-----------------------------------------------------------Wait For User Interaction----------------------------------------------------------------*)
	31550:
			IF	StepActionImpulse
				THEN
					NextStepPulse	:=	TRUE;
			END_IF;

			IF	StepAction AND
				( RTrigNextStep.Q OR
				ContinousMode )
				THEN
					IF CbaLimit
						THEN
							ZAxisLimitPos	:=	FALSE;
							ZaxisCbaLimit	:=	TRUE;
							StepNew			:= 	10;
							NextStepPulse	:=	FALSE;
							StopChipBreaker	:=	TRUE;
							KeyNextStep		:=	FALSE;
							CbaLimit			:=	FALSE;
						ELSE
							IF	WarningAaxis
								THEN
									WarningAaxisIsSlow	:=	TRUE;	;
							END_IF;
							IF	CbaSpindleLowSpeed
								THEN
									CbaSpindleLowSpeedOutput	:=	TRUE;
							END_IF;
							ZaxisCbaLimit	:=	FALSE;
							StepNew			:= 	10;
							NextStepPulse	:=	FALSE;
							StopChipBreaker	:=	TRUE;
							KeyNextStep		:=	FALSE;
					END_IF;
			END_IF;

		(*--------------------------------------------------------------------Deactivate Axis---------------------------------------------------------------------*)

	31600 :
			(*Action*)
			IF	StepActionImPulse
				THEN
				(* set axis state for check *)
					AxisState	:=	STATE_DISABLED;
					(*X-Axis*)
					AxisCtrl[AxisNo.XAxis].Command.OperationMode.CmdPowerOn						:=	FALSE;
					AxisCtrl[AxisNo.XAxis].Command.OperationMode.CmdMoveAbsolut					:=	FALSE;
					AxisCtrl[AxisNo.XAxis].Command.OperationMode.CmdJog							:=	FALSE;
					AxisCtrl[AxisNo.XAxis].Command.OperationMode.CmdJogHandwheel					:=	FALSE;
				(* Reset z-axis *)
					AxisCtrl[AxisNo.ZAxis].Command.OperationMode.CmdPowerOn						:=	FALSE;
					AxisCtrl[AxisNo.ZAxis].Command.OperationMode.CmdMoveAbsolut					:=	FALSE;
					AxisCtrl[AxisNo.ZAxis].Command.OperationMode.CmdJog							:=	FALSE;
					AxisCtrl[AxisNo.ZAxis].Command.OperationMode.CmdJogHandwheel					:=	FALSE;
					(* Reset Y-axis *)
					AxisCtrl[AxisNo.YAxis].Command.OperationMode.CmdPowerOn						:=	FALSE;
					AxisCtrl[AxisNo.YAxis].Command.OperationMode.CmdMoveAbsolut					:=	FALSE;
					AxisCtrl[AxisNo.YAxis].Command.OperationMode.CmdJog							:=	FALSE;
					AxisCtrl[AxisNo.YAxis].Command.OperationMode.CmdJogHandwheel					:=	FALSE;

					MachineCtrl.Peripheral.ChipBreaker.Auto.DustFan.CmdOn							:=	FALSE;
					MachineCtrl.Peripheral.ChipBreaker.Auto.LowSpeedMonitoring.IsDeactivated			:=	FALSE;
			END_IF;

			(* transition *)
			IF	StepAction AND
				(NOT StepActionImPulse) AND
				(* all axis are disabled *)
					Axis[AxisNo.XAxis].Status.Disabled  AND
					Axis[AxisNo.ZAxis].Status.Disabled AND
					Axis[AxisNo.YAxis].Status.Disabled
				THEN
					StepNew	:= 31610;							(* -> Activate Safety State*)
			END_IF;
		(* ----------------------------------------------------------------------- Activate Safety State-----------------------------------------------------------------------*)
	31610:
			(*Action*)
			IF	StepActionImPulse
				THEN
					MachineCtrl.Peripheral.ChipBreaker.Auto.DustFan.CmdOn			:=	FALSE;
					MachineCtrl.Peripheral.SafetyState.CmdActivate					:=	TRUE;
					MachineCtrl.Peripheral.ExternalControl.StatusLedOnTouch1			:=	FALSE;
					MachineCtrl.Peripheral.ExternalControl.StatusLedOnTouch2			:=	FALSE;
			END_IF;

			(*Transition*)
			IF	StepAction AND
			(NOT StepActionImPulse) AND
			( NOT MachineCtrl.Peripheral.SafetyState.CmdDeactivate ) AND
			MachineCtrl.state.SafetyState.unit.IsActive
			THEN
					MachineCtrl.Peripheral.ChipBreaker.Auto.LowSpeedMonitoring.IsDeactivated		:=	FALSE;
					MachineCtrl.ProcessControl.Event.En											:=	FALSE;
					StopChipBreaker	:=	TRUE;
					StepNew	:= 0;
			END_IF;

		(*#######################################END-Stop_Process#################################################*)

	END_CASE;

		ACT_Pneumatic();
		ACT_Stepper();


	ACT_TIME();

	StepperResults(
					sNetId					:=	'' ,
					sPathName				:= 	'C:\Loroch.UI\Beckhoff\StepperResults',
					FileName				:= 	'CbaStepperResults',
					FileNameExtension		:=	FileNameExtension ,
					bExecute				:= 	StartWriting,
					StartTime				:=	stTimeStartM ,
					EndTime					:=	stTimeEndM ,
					SawBladeWidth			:=	UI.Order.SawBlade.Width ,
					ZaxisStartPos				:=	ZPosition,
					MeasurmentFailed		:=	'' ,
					NominalRefPosition		:= 	AaxisRefPosTemp,
					Duration					:=	DurationAaxisMotion ,
					EdgeFront				:=	(*MarginFrontValue ,*)SecondEdge,
					EdgeRear				:=	(*MarginRearValue ,*)AaxisRefPosTemp,
					ZaxisTouchPosition		:=	ZposForCsv ,
					Busy					=> ,
					Error					=> ,
					ErrId					=> 			);






























































          

ACTION ACT_Pneumatic:
                

CASE	SfcChipBreakerAuto.Step	OF

	(*-----------------------------------------------------Transition Pneumatic Cylinder-10------------------------------------------------------*)
	990	:		(*Transition*)
					IF 	ChipBreakerFr
						THEN
							StepNew		:=	1000;			(*ChipBreakerFront With Pneumatic Cylindre *)
						ELSIF	ChipBreakerRe AND
								(NOT ChipBreakerFr)
						THEN
							StepNew			:=	1100;		(*ChipBreaker Rear  With Pneumatic Cylindre *)
							NumberTouch	:=	0;			(*Init number of touch to 0*)
					END_IF;
	(*--------------------------------------------------------ChipBreakerFront With Cylindre --------------------------------------------------------*)
	1000	:		(*Action*)
					IF 	StepActionImpulse AND
						(NOT MachineCtrl.State.ChipBreaker.Auto.TurbinePosition.InFrontPosition)
						THEN
							IF	NOT UI.MachineSpecification.Base.DemoMode
								THEN
									MachineCtrl.Peripheral.ChipBreaker.Auto.TurbinePosition.CmdBackward	:=	FALSE;
									MachineCtrl.Peripheral.ChipBreaker.Auto.TurbinePosition.CmdForward	:=	TRUE;
							END_IF;
					END_IF;
					(*Transition*)
					IF 	StepAction AND
						(NOT StepActionImpulse) AND
						(NOT MachineCtrl.Peripheral.ChipBreaker.Auto.TurbinePosition.CmdForward) AND
						( MachineCtrl.State.ChipBreaker.Auto.TurbinePosition.InFrontPosition OR
						UI.MachineSpecification.Base.DemoMode)
						THEN
							StepNew		:=	1010;			(*Move Z-Axis Up *)
					END_IF;
	(*------------------------------------------------------------Wait For User Interaction---------------------------------------------------------------*)
	1010:			(*Action*)
					IF	StepActionImpulse
						THEN
							NextStepPulse	:=	TRUE;
					END_IF;
					(*Transition*)
					IF	StepAction AND
						( RTrigNextStep.Q OR
						ContinousMode )
						THEN
							StepNew			:= 	1220;		(*Move Z-Axis Up *)
							NextStepPulse	:=	FALSE;
					END_IF;
	(*----------------------------------------------------------Wait For User Interaction---------------------------------------------------------------*)
	1100:			(*Action*)
					IF	StepActionImpulse
						THEN
							NextStepPulse	:=	TRUE;
					END_IF;
					(*Transition*)
					IF	StepAction AND
						( RTrigNextStep.Q OR
						ContinousMode )
						THEN
							StepNew			:= 	1110;
							NextStepPulse	:=	FALSE;
					END_IF;
END_CASE;

              
END_ACTION

ACTION ACT_Stepper:
                

CASE	SfcChipBreakerAuto.Step	OF

	(*-----------------------------------------------ChipBreakerRearPosUsingServoMotor------------------------------------------------*)
	975:			(*Action*)
				IF 	StepActionImpulse
					THEN
						AxisCtrl[AxisNo.AAxis].Command.OperationMode.CmdJog				:=	TRUE;
						AxisCtrl[AxisNo.AAxis].Command.ExternalControl.Override				:=	100;
						AxisCtrl[AxisNo.AAxis].Command.NominalValue.VeloJog				:=	0.3;
						IF	(MachineCtrl.State.ChipBreaker.Auto.AaxisActualPos <=  ARearPos)
							THEN
								AxisCtrl[AxisNo.AAxis].Command.ExternalControl.StartPlus		:=	FALSE;
								AxisCtrl[AxisNo.AAxis].Command.ExternalControl.StartMinus		:=	TRUE;
							ELSE
								AxisCtrl[AxisNo.AAxis].Command.ExternalControl.StartPlus		:=	TRUE;
								AxisCtrl[AxisNo.AAxis].Command.ExternalControl.StartMinus		:=	FALSE;
						END_IF;
				END_IF;
				(*Transition*)
				IF 	StepAction AND
					(NOT StepActionImpulse) AND
					(MachineCtrl.State.ChipBreaker.Auto.AaxisActualPos <=  (ARearPos +AaxisTolerenceSlow)) AND
					(MachineCtrl.State.ChipBreaker.Auto.AaxisActualPos >=  (ARearPos -AaxisTolerenceSlow))
					THEN
						AxisCtrl[AxisNo.AAxis].Command.ExternalControl.StartPlus			:=	FALSE;
						AxisCtrl[AxisNo.AAxis].Command.ExternalControl.StartMinus			:=	FALSE;		(*Stop Moving   A-Axis*)
						StepNew				:=	 1100;
						StartMonitoringAaxis	:=	FALSE;
				END_IF;
	(*-----------------------------------------------1: front------------------Wait For User Interaction----------------------------------------------------*)
	980:			(*Action*)
				IF	StepActionImpulse
					THEN
						NextStepPulse	:=	TRUE;
				END_IF;
				(*Transition*)
				IF	StepAction AND
					( RTrigNextStep.Q OR
					TestZ )
					THEN
						StartMonitoringAaxis	:=	TRUE;
						IF 	(MachineCtrl.State.ChipBreaker.Auto.AaxisActualPos <= AaxisRefPosTemp)
							THEN
								StepNew			:= 	981;  		(*Start moving in the negative direction in order to reach the reference position*)
								AaxisActPosition	:=	MachineCtrl.State.ChipBreaker.Auto.AaxisActualPos ;
								StartMovingStepByStepRear		:=	TRUE;
								StartMovingStepByStepFront		:=	FALSE;
							ELSE
								StepNew			:= 	9882;;		(*Start moving in the positive  direction in order to reach the reference position*)
								AaxisActPosition	:=	MachineCtrl.State.ChipBreaker.Auto.AaxisActualPos ;
								StartMovingStepByStepRear		:=	FALSE;
								StartMovingStepByStepFront		:=	TRUE;;
								AaxisRefPosTemp	:=	AaxisRefPosTemp - (0.5*UI.Order.SawBlade.Width);  (*0.2*)
								StepMotorDestination	:=	AaxisRefPosTemp;
						END_IF;
						StepMotorDestination	:=	AaxisRefPosTemp;
						AaxisActPosition		:=	 MachineCtrl.State.ChipBreaker.Auto.AaxisActualPos;
				END_IF;
	(*----------------------------------Action:Move A-Axis To Reference Position ,moving with minus : Backward ---------------------------------*)
	981:			(*Action*)
				IF 	StepActionImpulse
					THEN
						AxisCtrl[AxisNo.AAxis].Command.OperationMode.CmdJog					:=	TRUE;
						AxisCtrl[AxisNo.AAxis].Command.ExternalControl.Override				:=	100;
						AxisCtrl[AxisNo.AAxis].Command.NominalValue.VeloJog					:=	1;
						IF	(MachineCtrl.State.ChipBreaker.Auto.AaxisActualPos<=  AaxisRefPosTemp )
							THEN
								AxisCtrl[AxisNo.AAxis].Command.ExternalControl.StartPlus		:=	FALSE;;
								AxisCtrl[AxisNo.AAxis].Command.ExternalControl.StartMinus		:=	TRUE;;
							ELSE
								AxisCtrl[AxisNo.AAxis].Command.ExternalControl.StartPlus		:=	TRUE;;
								AxisCtrl[AxisNo.AAxis].Command.ExternalControl.StartMinus		:=	FALSE;;
						END_IF;
				END_IF;
				(*Transition*)
				IF 	StepAction AND
					(NOT  StepActionImpulse) AND
					(MachineCtrl.State.ChipBreaker.Auto.AaxisActualPos >=  (AaxisRefPosTemp- AaxisTolerenceFast)) AND
					(MachineCtrl.State.ChipBreaker.Auto.AaxisActualPos <=  ( AaxisRefPosTemp + AaxisTolerenceFast))
					THEN
						StepNew				:=		995;
						AxisCtrl[AxisNo.AAxis].Command.ExternalControl.StartPlus				:=	FALSE;
						AxisCtrl[AxisNo.AAxis].Command.ExternalControl.StartMinus				:=	FALSE;
						StartMonitoringAaxis	:=	FALSE;
						AaxisRefPosTemp	:=	MachineCtrl.State.ChipBreaker.Auto.AaxisActualPos - (0.5*UI.Order.SawBlade.Width);
						MonitoringTouchBack	:=	AaxisRefPosTemp - 0.01;
				END_IF;
	(*------------------------------------------------------move forward to make sure that the grindinfg whee will touch the sb----------------------*)
	995:			(*Transition*)
				IF	StepActionImpulse
					THEN
						NextStepPulse		:=	TRUE;
				END_IF;
				(*Transition*)
				IF	StepAction AND
					( RTrigNextStep.Q OR
					TestZ )
					THEN
						StepNew				:= 	996;				(* Moving stepper backward befor moving up Z-axis  *)
						NextStepPulse		:=	FALSE;
						StartMonitoringAaxis	:=	TRUE;
						StepMotorDestination	:=	AaxisRefPosTemp;
						AaxisActPosition		:=	 MachineCtrl.State.ChipBreaker.Auto.AaxisActualPos;
				END_IF;
	(*-----------------------------------------------Moving Stepper Backward before moving z-axis Up--------------------------------------------------*)
	996:
				(*Action*)
				IF 	StepActionImpulse
					THEN
						AxisCtrl[AxisNo.AAxis].Command.OperationMode.CmdJog				:=	TRUE;
						AxisCtrl[AxisNo.AAxis].Command.ExternalControl.Override				:=	100;
						AxisCtrl[AxisNo.AAxis].Command.NominalValue.VeloJog				:=	1;
						IF	(MachineCtrl.State.ChipBreaker.Auto.AaxisActualPos >=  AaxisRefPosTemp)
							THEN
								AxisCtrl[AxisNo.AAxis].Command.ExternalControl.StartPlus		:=	TRUE;;
								AxisCtrl[AxisNo.AAxis].Command.ExternalControl.StartMinus		:=	FALSE;;
							ELSE
								AxisCtrl[AxisNo.AAxis].Command.ExternalControl.StartPlus		:=	FALSE;;
								AxisCtrl[AxisNo.AAxis].Command.ExternalControl.StartMinus		:=	TRUE;;;
						END_IF;
				END_IF;
				(*Transition*)
				IF 	StepAction AND
					(NOT  StepActionImpulse) AND
					(MachineCtrl.State.ChipBreaker.Auto.AaxisActualPos >=  (AaxisRefPosTemp- AaxisTolerenceFast )) AND
					(MachineCtrl.State.ChipBreaker.Auto.AaxisActualPos <=  ( AaxisRefPosTemp + AaxisTolerenceFast ))
					THEN
						StepNew				:= 9810;
						AxisCtrl[AxisNo.AAxis].Command.ExternalControl.StartMinus				:=	FALSE;
						AxisCtrl[AxisNo.AAxis].Command.ExternalControl.StartPlus				:=	FALSE;
						StartMonitoringAaxis	:=	FALSE;
				END_IF;
	(*-------------------------------------------------------------------------find out the reference position ---------------------------------------------------------*)
	9810:		(* Action *)
				IF	StepActionImpulse
					THEN
						NextStepPulse	:=	TRUE;
				END_IF;
				(*Transition*)
				IF	StepAction AND
					( RTrigNextStep.Q OR
					ContinousMode )
					THEN
						StepNew			:= 	9815;				(* *)
						NextStepPulse	:=	FALSE;
				END_IF;
	(*----------------------------------------------------Move the Z axis up with touch probe active---------------------------------------------------*)
	9815:
				(*Action*)
				IF	StepActionImPulse
					THEN
						StartMonitoringAaxis	:=	FALSE;
						AxisCtrl[AxisNo.ZAxis].Command.OperationMode.CmdMoveAbsolut				:=	TRUE;
						AxisCtrl[AxisNo.ZAxis].Command.OperationMode.CmdMoveAbsolutTouchProbe	:=	TRUE;
						AxisCtrl[AxisNo.ZAxis].Command.NominalValue.VeloMoveAbsolut				:=	2;
						AxisCtrl[AxisNo.ZAxis].Command.NominalValue.PositionMoveAbsolut				:= 	Axis[AxisNo.ZAxis].NcToPlc.ActPos - 14;
				END_IF;
				(*Transition*)
				IF 	StepAction AND
					(NOT StepActionImPulse) AND
					(NOT AxisCtrl[AxisNo.ZAxis].Command.OperationMode.CmdMoveAbsolutTouchProbe )
					THEN
						IF	( AxisCtrl[AxisNo.ZAxis].Feedback.State.TouchProbe.ActiveAndAxisStopped)
							THEN
								TriesNumber	:=	TriesNumber +1 ;

								ZTouchPos				:=	Axis[AxisNo.ZAxis].NcToPlc.ActPos;
								IF	(TriesNumber = 1)
									THEN
										ZTouchPosFirstTouchPos	:=	ZTouchPos;
										ZNoTouch				:=	ZTouchPosFirstTouchPos - 1;  (*0.3*)
										ZposForCsv				:=	ZTouchPosFirstTouchPos;
								END_IF;

								AxisCtrl[AxisNo.ZAxis].Command.OperationMode.CmdMoveAbsolut				:=	FALSE;
								AxisCtrl[AxisNo.ZAxis].Command.OperationMode.CmdMoveAbsolutTouchProbe	:=	FALSE;
								StepNew			:=	9817;
						END_IF;
						(*Check of the touch number *)
						IF	(TriesNumber >=1)
							THEN
								StepNew						:=	9817;
								AaxisStepPositionIsReached	:=	TRUE;
								AxisCtrl[AxisNo.ZAxis].Command.OperationMode.CmdMoveAbsolut	:=	FALSE;
								LastZPos					:=	Axis[AxisNo.ZAxis].NcToPlc.ActPos ;
						END_IF;
						(*if no touch detected --> Warning  *)
						IF	(Axis[AxisNo.ZAxis].NcToPlc.ActPos <  LimitZaxis)
							THEN
								StepNew		:=	6000;;						(*If There is No Touch --> ERROR*)
								MachineCtrl.ProcessControl.Warning.No		:=	PSM_Fault_ErrorChipBreakerAuto;
								MachineCtrl.ProcessControl.Warning.En		:=	TRUE;
								MachineCtrl.Peripheral.Buzzer.Unit.CmdOn	:=	TRUE;
								MachineCtrl.ProcessControl.Warning.Data		:=	'';
						END_IF;
				END_IF;
	(*---------------------------------------------------------------------Wait for User Interaction-----------------------------------------------------------------------*)
	9817:
				(*Action*)
				IF	StepActionImpulse
					THEN
						NextStepPulse	:=	TRUE;
						AxisCtrl[AxisNo.ZAxis].Command.OperationMode.CmdMoveAbsolut	:=	FALSE;
				END_IF;
				(*Transition*)
				IF	StepAction AND
					(NOT StepActionImPulse)
					THEN
						StepNew			:=	9819;
				END_IF;
	(*----------------------------------------------------------------Move Z axis down 0,5MM----------------------------------------------------------------------------*)
	9819:
				(*Action*)
				IF 	StepActionImPulse
					THEN
						AxisState																:=	STATE_WAIT_NEWOPERATION;
						AxisCtrl[AxisNo.ZAxis].Command.OperationMode.CmdMoveAbsolut				:=	TRUE;
						AxisCtrl[AxisNo.ZAxis].Command.ExternalControl.override						:=	100;
						AxisCtrl[AxisNo.ZAxis].Command.OperationMode.CmdMoveAbsolutTouchProbe	:=	FALSE;		(*Down without Touch Probe :to not affect the touchnumber  *)
						AxisCtrl[AxisNo.ZAxis].Command.NominalValue.PositionMoveAbsolut				:=	ZTouchPosFirstTouchPos	+ 0.5;
						AxisCtrl[AxisNo.ZAxis].Command.NominalValue.VeloMoveAbsolut				:=	3;
				END_IF;
				(*Transition*)
				IF	StepAction AND
					NOT StepActionImPulse  AND
					(* status z-axis *)
					( NOT Axis[AxisNo.ZAxis].Status.Disabled ) AND
					Axis[AxisNo.ZAxis].Status.InTargetPosition AND
					Axis[AxisNo.ZAxis].Status.StandStill	AND
					( NOT AxisCtrl[AxisNo.ZAxis].Command.OperationMode.CmdMoveAbsolut )AND
					( AxisCtrl[AxisNo.ZAxis].feedback.state.ActualFbState = AxisState )
					THEN
						AxisCtrl[AxisNo.ZAxis].Command.OperationMode.CmdMoveAbsolut	:=	FALSE;
						StepNew		:=	9821;
				END_IF;
	(*----------------------------------------------Wait for User Interacton-----------------------------------------------------------------------*)
	9821:		(*Transition*)
				IF	RTrigNextStep.Q  OR
					TestZ
					THEN
						StepNew	:=	9822;
						AaxisRefPosTemp	:=	7 ;
						StartMonitoringAaxis	:=	TRUE;
						StepMotorDestination	:=	AaxisRefPosTemp;
						AaxisActPosition		:=	 MachineCtrl.State.ChipBreaker.Auto.AaxisActualPos;
				END_IF;
	(*----------------------------------------------------------Move A Axis Backward-----------------------------------------------------*)
	9822:
				(*Action*)
				IF 	StepActionImpulse
					THEN
						AxisCtrl[AxisNo.AAxis].Command.OperationMode.CmdJog				:=	TRUE;
						AxisCtrl[AxisNo.AAxis].Command.ExternalControl.Override				:=	100;
						AxisCtrl[AxisNo.AAxis].Command.NominalValue.VeloJog				:=	1;
						IF	(MachineCtrl.State.ChipBreaker.Auto.AaxisActualPos <=7)
							THEN
								AxisCtrl[AxisNo.AAxis].Command.ExternalControl.StartPlus				:=	FALSE;
								AxisCtrl[AxisNo.AAxis].Command.ExternalControl.StartMinus				:=	TRUE;;
							ELSE
								AxisCtrl[AxisNo.AAxis].Command.ExternalControl.StartPlus				:=	TRUE;
								AxisCtrl[AxisNo.AAxis].Command.ExternalControl.StartMinus				:=	FALSE;;
						END_IF;
				END_IF;
				(*Transition*)
				IF 	StepAction AND
					(NOT  StepActionImpulse) AND
					(MachineCtrl.State.ChipBreaker.Auto.AaxisActualPos >=  (AaxisRefPosTemp- AaxisTolerenceFast)) AND
					(MachineCtrl.State.ChipBreaker.Auto.AaxisActualPos <=  ( AaxisRefPosTemp + AaxisTolerenceFast))
					THEN
						StepNew				:=		5000;
						AxisCtrl[AxisNo.AAxis].Command.ExternalControl.StartPlus				:=	FALSE;
						AxisCtrl[AxisNo.AAxis].Command.ExternalControl.StartMinus				:=	FALSE;
						StartMonitoringAaxis	:=	FALSE;
				END_IF;
	(*---------------------------------------------------------Move Z-Axis to Z-No Touch Position-------------------------------------------*)
	5000:
				(*Transition*) (*wait for new operation*)
				IF	RTrigNextStep.Q OR
					TestZ
					THEN
						StepNew		:=	5010;
				END_IF;
	(*----------------------------------------------------------------Move Z-Axis To No touch Position -------------------------------------*)
	5010:		(*Action*)
				IF 	StepActionImPulse
					THEN
						AxisState											:=	STATE_WAIT_NEWOPERATION;
						AxisCtrl[AxisNo.ZAxis].Command.OperationMode.CmdMoveAbsolut					:=	TRUE;
						AxisCtrl[AxisNo.ZAxis].Command.ExternalControl.override						:=	100;
						AxisCtrl[AxisNo.ZAxis].Command.OperationMode.CmdMoveAbsolutTouchProbe				:=	TRUE;
						AxisCtrl[AxisNo.ZAxis].Command.NominalValue.PositionMoveAbsolut					:=	ZNoTouch;
						AxisCtrl[AxisNo.ZAxis].Command.NominalValue.VeloMoveAbsolut					:=	0.25;
				END_IF;
				(*Transition*)
				IF	StepAction AND
					NOT StepActionImPulse  AND
					(* status z-axis *)
					( NOT Axis[AxisNo.ZAxis].Status.Disabled ) AND
					Axis[AxisNo.ZAxis].Status.InTargetPosition AND
					Axis[AxisNo.ZAxis].Status.StandStill	AND
					( NOT AxisCtrl[AxisNo.ZAxis].Command.OperationMode.CmdMoveAbsolut )AND
					( AxisCtrl[AxisNo.ZAxis].feedback.state.ActualFbState = AxisState )
					THEN
						AxisCtrl[AxisNo.ZAxis].Command.OperationMode.CmdMoveAbsolut	:=	FALSE;
						StepNew		:=	5020;
				END_IF;

				IF 	StepAction AND
					(NOT StepActionImPulse) AND
					(NOT AxisCtrl[AxisNo.ZAxis].Command.OperationMode.CmdMoveAbsolutTouchProbe )
					THEN
						IF	( AxisCtrl[AxisNo.ZAxis].Feedback.State.TouchProbe.ActiveAndAxisStopped)
							THEN
								StepNew		:=	6000;;						(*If There is No Touch --> ERROR*)
								MachineCtrl.ProcessControl.Warning.No		:=	EvUnexpectedTouchWithZAxis ;
								MachineCtrl.ProcessControl.Warning.En		:=	TRUE;
								MachineCtrl.Peripheral.Buzzer.Unit.CmdOn	:=	TRUE;
								MachineCtrl.ProcessControl.Warning.Data		:=	'';
						END_IF;
				END_IF;

	(*---------------------------------------------------------------Wait For User Interaction---------------------------------------------------*)
	5020:		(*Transition*)
				IF	RTrigNextStep.Q  OR
					TREU
					THEN
						StepNew				:=	5030;
						StartMonitoringAaxis	:=	TRUE;
						AaxisActPosition		:=	 MachineCtrl.State.ChipBreaker.Auto.AaxisActualPos;
				END_IF;
	(*-----------------------------------------------------------------Move A-Axis Forward ---------------------------------------*)
	5030:		(*Action*)
				IF 	StepActionImpulse
					THEN
						AxisCtrl[AxisNo.AAxis].Command.OperationMode.CmdJog						:=	TRUE;
						AxisCtrl[AxisNo.AAxis].Command.ExternalControl.Override						:=	100;
						AxisCtrl[AxisNo.AAxis].Command.NominalValue.VeloJog						:=	0.1;
						AxisCtrl[AxisNo.AAxis].Command.ExternalControl.StartPlus						:=	TRUE;
						AxisCtrl[AxisNo.AAxis].Command.ExternalControl.StartMinus						:=	FALSE;;
				END_IF;

				RTrigMonitoringCrash(CLK:=( MachineCtrl.State.ChipBreaker.Auto.AaxisActualPos <MonitoringTouchBack) , Q=> );
				(*Transition*)
				IF	MachineCtrl.State.TouchSensor.Machine.IsActuated(*MachineCtrl.State.ChipBreaker.Auto.CrashSignalDetected*)
					THEN
						AxisCtrl[AxisNo.AAxis].Command.ExternalControl.StartPlus						:=	FALSE;
						AxisCtrl[AxisNo.AAxis].Command.ExternalControl.StartMinus						:=	FALSE;
						AxisCtrl[AxisNo.ZAxis].Command.OperationMode.CmdMoveAbsolut				:=	FALSE;
						AxisCtrl[AxisNo.ZAxis].Command.OperationMode.CmdMoveAbsolutTouchProbe	:=	FALSE;
						AaxisRefPosTemp	:=	 MachineCtrl.State.ChipBreaker.Auto.AaxisActualPos;		(*First Edge Position*)
						FirstEdgePos			:=	 MachineCtrl.State.ChipBreaker.Auto.AaxisActualPos;
						StepNew				:=	5035;
						StartMonitoringAaxis	:=	FALSE;
						RTrigMonitoringCrash(CLK:= FALSE);
				END_IF;

				(*New Monitoring *)
				IF	RTrigMonitoringCrash.Q AND
					(NOT MachineCtrl.State.TouchSensor.Machine.IsActuated)
					THEN
						StepNew		:=	6000;;						(*If There is No Touch --> ERROR*)
						MachineCtrl.ProcessControl.Warning.No		:=	EvNoTouchSignalDetected;
						MachineCtrl.ProcessControl.Warning.En		:=	TRUE;
						MachineCtrl.Peripheral.Buzzer.Unit.CmdOn	:=	TRUE;
						MachineCtrl.ProcessControl.Warning.Data		:=	'';
				END_IF;
	(*--------------------------------------------------------------------------Wait For User Interaction----------------------------------------------------------------------*)
	5035:		(*Transition*)
				IF	RTrigNextStep.Q OR
					TestZ
					THEN
						StepNew		:=	5040;
						FirstEdgePos	:=	FirstEdgePos	+ 0.3;
						StartMonitoringAaxis	:=	TRUE;
						StepMotorDestination	:=	FirstEdgePos;
						AaxisActPosition		:=	 MachineCtrl.State.ChipBreaker.Auto.AaxisActualPos;
				END_IF;
	(*------------------------------------------------------------------------------Move a-Axis Backwars before To Move Z-Axis Dwn---------------------------------------*)
	5040:		(*Action*)
				IF 	StepActionImpulse
					THEN
						AxisCtrl[AxisNo.AAxis].Command.OperationMode.CmdJog				:=	TRUE;
						AxisCtrl[AxisNo.AAxis].Command.ExternalControl.Override				:=	100;
						AxisCtrl[AxisNo.AAxis].Command.NominalValue.VeloJog				:=	1;
						IF	(MachineCtrl.State.ChipBreaker.Auto.AaxisActualPos <= FirstEdgePos)
							THEN
								AxisCtrl[AxisNo.AAxis].Command.ExternalControl.StartPlus				:=	FALSE;
								AxisCtrl[AxisNo.AAxis].Command.ExternalControl.StartMinus				:=	TRUE;;
							ELSE
								AxisCtrl[AxisNo.AAxis].Command.ExternalControl.StartPlus				:=	TRUE;
								AxisCtrl[AxisNo.AAxis].Command.ExternalControl.StartMinus				:=	FALSE;;
						END_IF;
				END_IF;
				(*Transition*)
				IF 	StepAction AND
					(NOT  StepActionImpulse) AND
					(MachineCtrl.State.ChipBreaker.Auto.AaxisActualPos >=  (FirstEdgePos- AaxisTolerenceFast)) AND
					(MachineCtrl.State.ChipBreaker.Auto.AaxisActualPos <=  ( FirstEdgePos + AaxisTolerenceFast))
					THEN
						StepNew				:=		5045;
						AxisCtrl[AxisNo.AAxis].Command.ExternalControl.StartPlus				:=	FALSE;
						AxisCtrl[AxisNo.AAxis].Command.ExternalControl.StartMinus				:=	FALSE;
						StartMonitoringAaxis	:=	FALSE;
				END_IF;
	(*-----------------------------------------------------------------------------Z Dwn-----------------------------------------------------------------------------------------------*)
	5045:
				(*Action*)
				IF 	StepActionImPulse
					THEN
						AxisState																:=	STATE_WAIT_NEWOPERATION;
						AxisCtrl[AxisNo.ZAxis].Command.OperationMode.CmdMoveAbsolut				:=	TRUE;
						AxisCtrl[AxisNo.ZAxis].Command.ExternalControl.override						:=	100;
						AxisCtrl[AxisNo.ZAxis].Command.OperationMode.CmdMoveAbsolutTouchProbe	:=	FALSE;
						AxisCtrl[AxisNo.ZAxis].Command.NominalValue.PositionMoveAbsolut				:=	ZTouchPosFirstTouchPos 	+ 0.5;
						AxisCtrl[AxisNo.ZAxis].Command.NominalValue.VeloMoveAbsolut				:=	2;
				END_IF;
				(*Transition*)
				IF	StepAction AND
					NOT StepActionImPulse  AND
					(* status z-axis *)
					( NOT Axis[AxisNo.ZAxis].Status.Disabled ) AND
					Axis[AxisNo.ZAxis].Status.InTargetPosition AND
					Axis[AxisNo.ZAxis].Status.StandStill	AND
					( NOT AxisCtrl[AxisNo.ZAxis].Command.OperationMode.CmdMoveAbsolut )AND
					( AxisCtrl[AxisNo.ZAxis].feedback.state.ActualFbState = AxisState )
					THEN
						AxisCtrl[AxisNo.ZAxis].Command.OperationMode.CmdMoveAbsolut	:=	FALSE;
						StepNew		:=	5050;
				END_IF;
	(*--------------------------------------------------------------------------------------------------------------------*)
	5050:		(*---Transition----*)
				IF	RTrigNextStep.Q  OR
					TestZ
					THEN
						StepNew		:=	5060	;
						SecondEdge	:=	AaxisRefPosTemp
										- UI.Order.SawBlade.Width - 0.5(*1*);
						MonitoringTouchFront	:=	AaxisRefPosTemp -
												UI.Order.SawBlade.Width + 0.3 + 0.01;
						StartMonitoringAaxis	:=	TRUE; ;
						StepMotorDestination	:=	SecondEdge;
						AaxisActPosition		:=	 MachineCtrl.State.ChipBreaker.Auto.AaxisActualPos;
				END_IF;
	(*---------------------------------------A-Axis to front Position -------------------------------------------*)
	5060:		(*Action*)
				IF 	StepActionImpulse
					THEN
						AxisCtrl[AxisNo.AAxis].Command.OperationMode.CmdJog				:=	TRUE;
						AxisCtrl[AxisNo.AAxis].Command.ExternalControl.Override				:=	100;
						AxisCtrl[AxisNo.AAxis].Command.NominalValue.VeloJog				:=	1; ;
						IF	(MachineCtrl.State.ChipBreaker.Auto.AaxisActualPos >=  (SecondEdge))
							THEN
								AxisCtrl[AxisNo.AAxis].Command.ExternalControl.StartPlus				:=	TRUE;
								AxisCtrl[AxisNo.AAxis].Command.ExternalControl.StartMinus				:=	FALSE;;
							ELSE
								AxisCtrl[AxisNo.AAxis].Command.ExternalControl.StartPlus				:=	FALSE;
								AxisCtrl[AxisNo.AAxis].Command.ExternalControl.StartMinus				:=	TRUE;;
						END_IF;
				END_IF;
				(*Transition*)
				IF 	StepAction AND
					(NOT  StepActionImpulse) AND
					(MachineCtrl.State.ChipBreaker.Auto.AaxisActualPos >=  (SecondEdge- AaxisTolerenceFast)) AND
					(MachineCtrl.State.ChipBreaker.Auto.AaxisActualPos <=  ( SecondEdge + AaxisTolerenceFast))
					THEN
						StepNew				:=		5070;
						AxisCtrl[AxisNo.AAxis].Command.ExternalControl.StartPlus				:=	FALSE;
						AxisCtrl[AxisNo.AAxis].Command.ExternalControl.StartMinus				:=	FALSE;
						StartMonitoringAaxis	:=	FALSE;
				END_IF;
	(*-----------------------------------------------------Wait For User Interaction--------------------------------------------------------*)
	5070:		(*Transition*)
				IF	RTrigNextStep.Q OR
					TestZ
					THEN
						StepNew		:=	5080;
				END_IF;
	(*-------------------------------------------------------Z-Axis To No Touch Position-----------------------------------------------*)
	5080:		(*Transition*)
				IF 	StepActionImPulse
					THEN
						AxisState																:=	STATE_WAIT_NEWOPERATION;
						AxisCtrl[AxisNo.ZAxis].Command.OperationMode.CmdMoveAbsolut				:=	TRUE;
						AxisCtrl[AxisNo.ZAxis].Command.ExternalControl.override						:=	100;
						AxisCtrl[AxisNo.ZAxis].Command.OperationMode.CmdMoveAbsolutTouchProbe	:=	TRUE;		(*Down without Touch Probe :to not affect the touchnumber  *)
						AxisCtrl[AxisNo.ZAxis].Command.NominalValue.PositionMoveAbsolut				:=	ZNoTouch;
						AxisCtrl[AxisNo.ZAxis].Command.NominalValue.VeloMoveAbsolut				:=	0.25;
				END_IF;
				(*Transition*)
				IF	StepAction AND
					NOT StepActionImPulse  AND
					(* status z-axis *)
					( NOT Axis[AxisNo.ZAxis].Status.Disabled ) AND
					Axis[AxisNo.ZAxis].Status.InTargetPosition AND
					Axis[AxisNo.ZAxis].Status.StandStill	AND
					( NOT AxisCtrl[AxisNo.ZAxis].Command.OperationMode.CmdMoveAbsolut )AND
					( AxisCtrl[AxisNo.ZAxis].feedback.state.ActualFbState = AxisState )
					THEN
						AxisCtrl[AxisNo.ZAxis].Command.OperationMode.CmdMoveAbsolut	:=	FALSE;
						StepNew		:=	5090;
				END_IF;

				(*Error Monitoring*)
				IF 	StepAction AND
					(NOT StepActionImPulse) AND
					(NOT AxisCtrl[AxisNo.ZAxis].Command.OperationMode.CmdMoveAbsolutTouchProbe )
					THEN
						IF	( AxisCtrl[AxisNo.ZAxis].Feedback.State.TouchProbe.ActiveAndAxisStopped)
							THEN
								StepNew		:=	6000;;						(*If There is No Touch --> ERROR*)
								MachineCtrl.ProcessControl.Warning.No		:=	EvUnexpectedTouchWithZAxis;
								MachineCtrl.ProcessControl.Warning.En		:=	TRUE;
								MachineCtrl.Peripheral.Buzzer.Unit.CmdOn	:=	TRUE;
								MachineCtrl.ProcessControl.Warning.Data		:=	'';
						END_IF;
				END_IF;

	(*----------------------------------------------------Wait For User Interaction--------------------------------------------------------*)
	5090:		(*Transition*)
				IF	RTrigNextStep.Q OR
					TestZ
					THEN
						StepNew	:=	5100;		(*Move A-Axis Backward till touch with the SB*)
						StartMonitoringAaxis	:=	TRUE;
				END_IF;
	(*----------------------------------------Move A-Axis Backward till touch with the SB-----------------------------------------*)
	5100:		(*Action*)
				IF 	StepActionImpulse
					THEN
						AxisCtrl[AxisNo.AAxis].Command.OperationMode.CmdJog						:=	TRUE;
						AxisCtrl[AxisNo.AAxis].Command.ExternalControl.Override						:=	100;
						AxisCtrl[AxisNo.AAxis].Command.NominalValue.VeloJog						:=	0.1;
						AxisCtrl[AxisNo.AAxis].Command.ExternalControl.StartPlus						:=	FALSE;
						AxisCtrl[AxisNo.AAxis].Command.ExternalControl.StartMinus						:=	TRUE;;
					(*	StartMonitoringAaxis	:=	FALSE;*)
				END_IF;

				RTrigMonitoringCrash(CLK:= MachineCtrl.State.ChipBreaker.Auto.AaxisActualPos >=
																					 MonitoringTouchFront , Q=> );
				(*Transition*)
				IF	MachineCtrl.State.TouchSensor.Machine.IsActuated (*MachineCtrl.State.ChipBreaker.Auto.CrashSignalDetected*)
					THEN
						AxisCtrl[AxisNo.AAxis].Command.ExternalControl.StartPlus						:=	FALSE;
						AxisCtrl[AxisNo.AAxis].Command.ExternalControl.StartMinus						:=	FALSE;
						AxisCtrl[AxisNo.ZAxis].Command.OperationMode.CmdMoveAbsolut				:=	FALSE;
						AxisCtrl[AxisNo.ZAxis].Command.OperationMode.CmdMoveAbsolutTouchProbe	:=	FALSE;
						SecondEdge			:=	 MachineCtrl.State.ChipBreaker.Auto.AaxisActualPos;
						StepNew				:=	5110;
						StartMonitoringAaxis	:=	FALSE;
						RTrigMonitoringCrash(CLK:= FALSE);
				END_IF;

				IF	RTrigMonitoringCrash.Q(* AND
					(NOT MachineCtrl.State.TouchSensor.Machine.IsActuated)  *)
					THEN
						StepNew		:=	6000;;						(*If There is No Touch --> ERROR*)
						MachineCtrl.ProcessControl.Warning.No		:=	EvNoTouchSignalDetected;
						MachineCtrl.ProcessControl.Warning.En		:=	TRUE;
						MachineCtrl.Peripheral.Buzzer.Unit.CmdOn	:=	TRUE;
						MachineCtrl.ProcessControl.Warning.Data		:=	'';
				END_IF;

	(*----------------------------------------------Wait for User Interaction---------------------------------*)
	5110:		(*Transition*)
				IF	RTrigNextStep.Q OR
					TestZ
					THEN
						StepNew	:=	5120;	(*A-Axis Forward 1 MM*)
						StartMonitoringAaxis	:=	TRUE;
						StepMotorDestination	:=	SecondEdge-1;
						AaxisActPosition		:=	 MachineCtrl.State.ChipBreaker.Auto.AaxisActualPos;
				END_IF;
	(*------------------------------------------------A-Axis Forward -------------------------------------------*)
	5120:		(*Action*)
				IF 	StepActionImpulse
					THEN
						AxisCtrl[AxisNo.AAxis].Command.OperationMode.CmdJog				:=	TRUE;
						AxisCtrl[AxisNo.AAxis].Command.ExternalControl.Override				:=	100;
						AxisCtrl[AxisNo.AAxis].Command.NominalValue.VeloJog				:=	1;
						AxisCtrl[AxisNo.AAxis].Command.ExternalControl.StartPlus				:=	TRUE;
						AxisCtrl[AxisNo.AAxis].Command.ExternalControl.StartMinus				:=	FALSE;;
				END_IF;
				(*Transition*)
				IF 	StepAction AND
					(NOT  StepActionImpulse) AND
					(MachineCtrl.State.ChipBreaker.Auto.AaxisActualPos >=  (SecondEdge-1 - AaxisTolerenceFast)) AND
					(MachineCtrl.State.ChipBreaker.Auto.AaxisActualPos <=  ( SecondEdge -1 + AaxisTolerenceFast))
					THEN
						StepNew				:=		5130;		(*Z-Axis Moving Dwn*)
						AxisCtrl[AxisNo.AAxis].Command.ExternalControl.StartPlus				:=	FALSE;
						AxisCtrl[AxisNo.AAxis].Command.ExternalControl.StartMinus				:=	FALSE;
						StartMonitoringAaxis	:=	FALSE;
				END_IF;
	(*------------------------------------Wait For User Interaction-----------------------------------*)
	5130:		(*Transition*)
				IF	RTrigNextStep.Q OR
					TestZ
					THEN
						StepNew		:=5140;
				END_IF;
	(*------------------------------------------------------------------Z-Axis Dwn 1 MM--------------------------*)
	5140:		(*Action*)
				IF 	StepActionImPulse
					THEN
						AxisState																:=	STATE_WAIT_NEWOPERATION;
						AxisCtrl[AxisNo.ZAxis].Command.OperationMode.CmdMoveAbsolut				:=	TRUE;
						AxisCtrl[AxisNo.ZAxis].Command.ExternalControl.override						:=	100;
						AxisCtrl[AxisNo.ZAxis].Command.OperationMode.CmdMoveAbsolutTouchProbe	:=	FALSE;
						AxisCtrl[AxisNo.ZAxis].Command.NominalValue.PositionMoveAbsolut				:=	ZTouchPosFirstTouchPos   	+ 0.5;
						AxisCtrl[AxisNo.ZAxis].Command.NominalValue.VeloMoveAbsolut				:=	2;
				END_IF;
				(*Transition*)
				IF	StepAction AND
					NOT StepActionImPulse  AND
					(* status z-axis *)
					( NOT Axis[AxisNo.ZAxis].Status.Disabled ) AND
					Axis[AxisNo.ZAxis].Status.InTargetPosition AND
					Axis[AxisNo.ZAxis].Status.StandStill	AND
					( NOT AxisCtrl[AxisNo.ZAxis].Command.OperationMode.CmdMoveAbsolut )AND
					( AxisCtrl[AxisNo.ZAxis].feedback.state.ActualFbState = AxisState )
					THEN
						AxisCtrl[AxisNo.ZAxis].Command.OperationMode.CmdMoveAbsolut	:=	FALSE;
						StepNew		:=	5150;
				END_IF;
	(*-------------------------------------Wait For User Interaction---------------------------------------*)
	5150:		(*Action*)
				IF	RTrigNextStep.Q OR
					TestZ
					THEN
						StepNew		:=	9830;	(*next step*)
				END_IF;
			//	if stepper


	(*############################Stop During Touching Process###############*)
	6000:
				IF 	StepActionImPulse
					THEN
						AxisState																:=	STATE_WAIT_NEWOPERATION;
						AxisCtrl[AxisNo.ZAxis].Command.OperationMode.CmdPowerOn					:=	TRUE;;
						AxisCtrl[AxisNo.ZAxis].Command.OperationMode.CmdMoveAbsolut				:=	TRUE;
						AxisCtrl[AxisNo.ZAxis].Command.ExternalControl.override						:=	100;
						AxisCtrl[AxisNo.ZAxis].Command.OperationMode.CmdMoveAbsolutTouchProbe	:=	FALSE;
						AxisCtrl[AxisNo.ZAxis].Command.NominalValue.PositionMoveAbsolut				:=	Axis[AxisNo.ZAxis].NcToPlc.ActPos + 5;
						AxisCtrl[AxisNo.ZAxis].Command.NominalValue.VeloMoveAbsolut				:=	2;
				END_IF;
				(*Transition*)
				IF	StepAction AND
					NOT StepActionImPulse  AND
					(* status z-axis *)
					( NOT Axis[AxisNo.ZAxis].Status.Disabled ) AND
					Axis[AxisNo.ZAxis].Status.InTargetPosition AND
					Axis[AxisNo.ZAxis].Status.StandStill	AND
					( NOT AxisCtrl[AxisNo.ZAxis].Command.OperationMode.CmdMoveAbsolut )AND
					( AxisCtrl[AxisNo.ZAxis].feedback.state.ActualFbState = AxisState )
					THEN
						AxisCtrl[AxisNo.ZAxis].Command.OperationMode.CmdMoveAbsolut	:=	FALSE;
						StepNew		:=	6005;
				END_IF
	(*-------------------------------------------------------------------Release clamping----------------------------------------------------------------*)
	6005:
		(*Action*)
			IF	StepActionImPulse AND
				(NOT MachineCtrl.State.ChipBreaker.Auto.Clamping.IsReleased)
				THEN
					MachineCtrl.Peripheral.ChipBreaker.Auto.Clamping.CmdClose	:=	FALSE;
					MachineCtrl.Peripheral.ChipBreaker.Auto.Clamping.CmdOpen	:=	TRUE;
			END_IF;

			(* transition:  *)
			IF	StepAction AND
				(NOT StepActionImPulse) AND
				MachineCtrl.State.ChipBreaker.Auto.Clamping.IsReleased
			THEN
					StepNew	:= 	27000;					(*Z Axis  down*)
			END_IF;

	(*##############################################Error Out###############################################*)
	27000:
				(*Action*)
				IF	 StepActionImPulse
					THEN
						MachineCtrl.Peripheral.ChipBreaker.Auto.DustFan.CmdOn			:=	FALSE;
						AxisCtrl[AxisNo.AAxis].Command.ExternalControl.StartPlus			:=	FALSE;
						AxisCtrl[AxisNo.AAxis].Command.ExternalControl.StartMinus			:=	FALSE;		(*Stop Moving   A-Axis*)
						ErrorOut			:=	TRUE;
				END_IF;
				(*Transition*)

				IF 	StepAction AND
					(NOT StepActionImPulse)
					THEN
							StepNew		:=	0;
							ErrorOut		:=	FALSE;
				END_IF;
	(*####################################################################*)

	(*---------------------------------------Check The Notch Position--------------------------------------*)
	9900:
				(*Transition*)
				IF	NOT StepActionImPulse  AND
					StepAction
					THEN
						IF	 (TriesNumber>0) AND
							(NOT AaxisStepPositionIsReached)
							THEN
								StepNew				:=	982;(*Move Forward*)
								AaxisRefPosTemp	:= 	MachineCtrl.State.ChipBreaker.Auto.AaxisActualPos;
							END_IF;
							IF	AaxisStepPositionIsReached
							THEN
								AaxisRefPosTemp	:=	 MachineCtrl.State.ChipBreaker.Auto.AaxisActualPos;
								StepNew				:=	9830;
						END_IF;
				END_IF;
	(*-----------------------------------------------Check the Notch position----------------------------------*)
	9823:
				(*Transition*)
				IF	NOT StepActionImPulse  AND
					StepAction
					THEN
						IF	 (TriesNumber>0) AND
							(NOT AaxisStepPositionIsReached)
							THEN
								StepNew				:=	9825;(*Move Backward*)
								AaxisActPosition		:=	MachineCtrl.State.ChipBreaker.Auto.AaxisActualPos;
						END_IF;
						IF	AaxisStepPositionIsReached
							THEN
								StepNew				:=	9830;
								AaxisRefPosTemp	:= MachineCtrl.State.ChipBreaker.Auto.AaxisActualPos;
						END_IF;
				END_IF;
	(*------------------------------------------------Wait for User  Interaction------------ -----------------------*)
	9825:		(*Action*)
				IF	StepActionImpulse
					THEN
						NextStepPulse	:=	TRUE;
				END_IF;
				IF	StepAction AND
					( RTrigNextStep.Q OR
					ContinousMode )
					THEN
						StepNew			:= 	982;		(* *)
						NextStepPulse	:=	FALSE;
				END_IF;
	(*------------------------------------------------------------------------------------------------------------------*)
	9830:		(* Transition *)
				IF	StepAction
					THEN
						AFrontPos			:=     	SecondEdge + MarginFrontValue + ChipBreakerAutoGWwidth    		     ;
						ARearPos			:=      AaxisRefPosTemp	 - MarginRearValue - ChipBreakerAutoGWwidth     ;
						stTimeStartM			:=	stTimeStruct;
						StartWriting			:=	TRUE;
						StepNew				:=	985;
						StartMonitoringAaxis	:=	TRUE;
						StepMotorDestination	:=	AFrontPos;
						AaxisActPosition		:=	 MachineCtrl.State.ChipBreaker.Auto.AaxisActualPos;
				END_IF;
	(*---------------------------------------------------------Move  A-Axis to Reference Position-------------------------------------------------------------------*)
	982:
				(*Action*)
				IF 	StepActionImpulse
					THEN
						AxisCtrl[AxisNo.AAxis].Command.OperationMode.CmdJog				:=	TRUE;
						AxisCtrl[AxisNo.AAxis].Command.ExternalControl.Override				:=	100;
						AxisCtrl[AxisNo.AAxis].Command.NominalValue.VeloJog				:=	0.5;
						AxisCtrl[AxisNo.AAxis].Command.ExternalControl.StartMinus				:=	TRUE;
						AxisCtrl[AxisNo.AAxis].Command.ExternalControl.StartPlus				:=	FALSE;;
						IF	(TriesNumber >0)
							THEN
								AaxisRefPosTemp	:=	MachineCtrl.State.ChipBreaker.Auto.AaxisActualPos + 0.05;
						END_IF ;
				END_IF;
				(*Transition*)
				IF 	StepAction AND
					(NOT  StepActionImpulse) AND
					(MachineCtrl.State.ChipBreaker.Auto.AaxisActualPos >=  (AaxisRefPosTemp- AaxisTolerenceSlow)) AND
					(MachineCtrl.State.ChipBreaker.Auto.AaxisActualPos <=  ( AaxisRefPosTemp + AaxisTolerenceSlow))
					THEN
						AxisCtrl[AxisNo.AAxis].Command.ExternalControl.StartMinus				:=	FALSE;
						AxisCtrl[AxisNo.AAxis].Command.ExternalControl.StartPlus				:=	FALSE;;
						StepNew			:=	983;
						StartWaitAaxis	:=	FALSE;;
				END_IF;
	(*---------------------------------------------------------Wait before moving the stepper--------------------------------------------------------------*)
	983:			(*Transition*)
				WaitForAaxis(IN:=	StartWaitAaxis , PT:=TIME#2s , Q=> , ET=> );
				IF	TRUE
					THEN
						StepNew			:=	9810;
						StartWaitAaxis	:=	FALSE;
				END_IF;
	(*---------------------------------------------Moving the stepper to Reference position-0,2MM ------------------------------------------------*)
	9882:		(*Action*)
				IF 	StepActionImpulse
					THEN
						AxisCtrl[AxisNo.AAxis].Command.OperationMode.CmdJog				:=	TRUE;
						AxisCtrl[AxisNo.AAxis].Command.ExternalControl.Override				:=	100;
						AxisCtrl[AxisNo.AAxis].Command.NominalValue.VeloJog				:=	0.5;
						IF	(MachineCtrl.State.ChipBreaker.Auto.AaxisActualPos >=  (AaxisRefPosTemp))
							THEN
								AxisCtrl[AxisNo.AAxis].Command.ExternalControl.StartPlus				:=	TRUE;
								AxisCtrl[AxisNo.AAxis].Command.ExternalControl.StartMinus				:=	FALSE;;
							ELSE
								AxisCtrl[AxisNo.AAxis].Command.ExternalControl.StartPlus				:=	FALSE;
								AxisCtrl[AxisNo.AAxis].Command.ExternalControl.StartMinus				:=	TRUE;;
						END_IF;
				END_IF;
				(*Transition*)
				IF 	StepAction AND
					(NOT  StepActionImpulse) AND
					(MachineCtrl.State.ChipBreaker.Auto.AaxisActualPos >=  (AaxisRefPosTemp- AaxisTolerenceSlow)) AND
					(MachineCtrl.State.ChipBreaker.Auto.AaxisActualPos <=  ( AaxisRefPosTemp + AaxisTolerenceSlow))
					THEN
						StepNew				:=	9810;
						AxisCtrl[AxisNo.AAxis].Command.ExternalControl.StartPlus				:=	FALSE;
						AxisCtrl[AxisNo.AAxis].Command.ExternalControl.StartMinus				:=	FALSE;;
						StartMonitoringAaxis	:=	FALSE;
				END_IF;
	(*-------------------------Move the A-Axis with a high velocity till it reaches the 80% of destination-----------------------*)
	9850:
				(*Action*)
				IF 	StepActionImpulse
					THEN
						AxisCtrl[AxisNo.AAxis].Command.OperationMode.CmdJog				:=	TRUE;
						AxisCtrl[AxisNo.AAxis].Command.ExternalControl.Override				:=	100;
						AxisCtrl[AxisNo.AAxis].Command.NominalValue.VeloJog				:=	1;
						AxisCtrl[AxisNo.AAxis].Command.ExternalControl.StartPlus				:=	TRUE;
						AxisCtrl[AxisNo.AAxis].Command.ExternalControl.StartMinus				:=	FALSE;
						StartMonitoringAaxis												:=	TRUE;
					END_IF;
				(*Transition*)
				IF 	StepAction AND
					(NOT  StepActionImpulse) AND
					(NOT AxisCtrl[AxisNo.AAxis].Command.OperationMode.CmdMoveAbsolut) AND
					(MachineCtrl.State.ChipBreaker.Auto.AaxisActualPos >=  (AFront80 - AaxisTolerenceSlow)) AND
					(MachineCtrl.State.ChipBreaker.Auto.AaxisActualPos <=  (AFront80 + AaxisTolerenceSlow))
					THEN
						StepNew		:=	985;
						AxisCtrl[AxisNo.AAxis].Command.ExternalControl.StartPlus				:=	FALSE;
				END_IF;
	(*----------------------------------------------Move A-Axis to the calculated Front position-------------------------------------*)
	985	:			(*Action*)
					IF 	StepActionImpulse
						THEN
							AxisCtrl[AxisNo.AAxis].Command.OperationMode.CmdJog				:=	TRUE;
							AxisCtrl[AxisNo.AAxis].Command.ExternalControl.Override				:=	100;
							AxisCtrl[AxisNo.AAxis].Command.NominalValue.VeloJog				:=	1;
							IF	(MachineCtrl.State.ChipBreaker.Auto.AaxisActualPos<= AFrontPos)
								THEN
									AxisCtrl[AxisNo.AAxis].Command.ExternalControl.StartPlus		:=	FALSE;
									AxisCtrl[AxisNo.AAxis].Command.ExternalControl.StartMinus		:=	TRUE;
								ELSE
									AxisCtrl[AxisNo.AAxis].Command.ExternalControl.StartPlus		:=	TRUE;
									AxisCtrl[AxisNo.AAxis].Command.ExternalControl.StartMinus		:=	FALSE;
							END_IF;
					END_IF;
					(*Transition*)
					IF 	StepAction AND
						(NOT  StepActionImpulse) AND
						(NOT AxisCtrl[AxisNo.AAxis].Command.OperationMode.CmdMoveAbsolut) AND

						(MachineCtrl.State.ChipBreaker.Auto.AaxisActualPos >=  (AFrontPos - AaxisTolerenceFast)) AND
						(MachineCtrl.State.ChipBreaker.Auto.AaxisActualPos <=  (AFrontPos + AaxisTolerenceFast))
					THEN
						StepNew				:=	 12200;
						NumberTouch		:=	0;
						AxisCtrl[AxisNo.AAxis].Command.ExternalControl.StartPlus		:=	FALSE;
						AxisCtrl[AxisNo.AAxis].Command.ExternalControl.StartMinus		:=	FALSE;
						StartMonitoringAaxis	:=	FALSE;
					END_IF;
	(*----------------------------------------------Calclation of the start position of X-Axis and Z-Axis------------------------------------*)
	12200:			(*Transition*)
					IF 	StepAction AND
						(NOT StepActionImpulse)
						THEN
							ZAxisStartPosition													:=	ZTouchPosFirstTouchPos +0.7;
							XAxisStartPosition													:=	Axis[AxisNo.XAxis].NcToPlc.ActPos;
							XAxisEndPos														:=	Axis[AxisNo.XAxis].NcToPlc.ActPos  + 360;
							AxisCtrl[AxisNo.ZAxis].Command.OperationMode.CmdMoveAbsolut		:=	FALSE;										(*End Moving Up of Z-Axis*)
							StepNew															:=	12450;
					END_IF;
	(*-------------------------------------------------------------Wait For User Interaction------------------------------------------------------*)
	12450:
					(*Transition*)
					IF	RTrigNextStep.Q OR
						ContinousMode
						THEN
							StepNew		:=	1280;		(*Move Axis X&Z To Start position*)
					END_IF;
END_CASE;

              
END_ACTION

ACTION ACT_TIME:
                fbGetTime(	NETID		:= 	'',			(* Beckhoff Rechner '10.22.2.7.1.1' mit eingestellter Zeit, anstatt Maschinen-PC *)
			START		:= 	( NOT fbGetTime.BUSY ) AND ( NOT fbGetTime.START ),
			TMOUT		:= 	DEFAULT_ADS_TIMEOUT,
			BUSY		=>	 ,
			ERR		=> 	,
			ERRID		=>	,
			TIMESTR	=> 	stTimestruct );
              
END_ACTION
END_FUNCTION_BLOCK
